      move_thread_flag_4306 = 0
      move_thread_han_4306 = run move_thread_4306()
      while (True):
        sleep(1.0E-10)
        if (move_thread_flag_4306 > 1):
          join move_thread_han_4306
          $ 4307 "Until (distance)"
          break
        end
        sync()
      end
      $ 4308 "Direction: Base Z-"
      global move_thread_flag_4308=0
      thread move_thread_4308():
        enter_critical
        move_thread_flag_4308 = 1
        local towardsPos=calculate_point_to_move_towards(p[0.0,0.0,0.0,0.0,0.0,0.0], [0.0,0.0,-1.0], 1000.0)
        movel(towardsPos, a=0.007, v=0.007)
        move_thread_flag_4308 = 2
        exit_critical
      end
      move_thread_flag_4308 = 0
      move_thread_han_4308 = run move_thread_4308()
      while (True):
        local targetTcpDirection=get_target_tcp_speed()
        local stepsToRetract=tool_contact(direction=targetTcpDirection)
        if (stepsToRetract > 0):
          kill move_thread_han_4308
          stopl(0.02)
          local backTrackMovement=get_actual_joint_positions_history(stepsToRetract)
          local contactPose=get_forward_kin(backTrackMovement)
          local posDir=[targetTcpDirection[0],targetTcpDirection[1],targetTcpDirection[2]]
          local retractTo=contactPose
          if (norm(posDir) > 1e-6):
            local normalizedPosDir=normalize(posDir)
            local additionalRetraction=p[normalizedPosDir[0] * 0.0, normalizedPosDir[1] * 0.0, normalizedPosDir[2] * 0.0, 0, 0, 0]
            retractTo = pose_sub(contactPose, additionalRetraction)
          end
          movel(retractTo, a=0.02, v=0.1)
          $ 4309 "Until (tool_contact_detection)"
          break
        end
        sync()
      end
      $ 4310 "Popup: punto contacto alanzdo"
      popup("punto contacto alanzdo", "Mensaje", False, False, blocking=True)
      $ 4311 "Direction: Base Z+"
      global move_thread_flag_4311=0
      thread move_thread_4311():
        enter_critical
        move_thread_flag_4311 = 1
        local towardsPos=calculate_point_to_move_towards(p[0.0,0.0,0.0,0.0,0.0,0.0], [0.0,0.0,1.0], 0.007)
        movel(towardsPos, a=0.015, v=0.015)
        move_thread_flag_4311 = 2
        exit_critical
      end
      move_thread_flag_4311 = 0
      move_thread_han_4311 = run move_thread_4311()
      while (True):
        sleep(1.0E-10)
        if (move_thread_flag_4311 > 1):
          join move_thread_han_4311
          $ 4312 "Until (distance)"
          break
        end
        sync()
      end
      $ 4313 "Wait: 0.3"
      sleep(0.3)
      $ 4314 "Set CO[1]=Encender"
      set_configurable_digital_out(1, True)
      $ 4315 "Wait: 0.3"
      sleep(0.3)
      $ 4316 "Loop 1 times"
      Loop_32 = 0
      while (Loop_32 < 1):
        $ 4317 "bajar≔pose_add(get_actual_tcp_pose(), bajada_broca)"
        global bajar= pose_add ( get_actual_tcp_pose (), bajada_broca)
        $ 4318 "bajar" "breakAfter"
        movel(bajar, a=0.004, v=0.004)
        $ 4319 "subir≔pose_sub(get_actual_tcp_pose(), bajada_broca)"
        global subir= pose_sub ( get_actual_tcp_pose (), bajada_broca)
        $ 4320 "Direction: Base Z+"
        global move_thread_flag_4320=0
        thread move_thread_4320():
          enter_critical
          move_thread_flag_4320 = 1
          local towardsPos=calculate_point_to_move_towards(p[0.0,0.0,0.0,0.0,0.0,0.0], [0.0,0.0,1.0], 0.002)
          movel(towardsPos, a=0.015, v=0.015)
          move_thread_flag_4320 = 2
          exit_critical
        end
        move_thread_flag_4320 = 0
        move_thread_han_4320 = run move_thread_4320()
        while (True):
          sleep(1.0E-10)
          if (move_thread_flag_4320 > 1):
            join move_thread_han_4320
            $ 4321 "Until (distance)"
            break
          end
          sync()
        end
        $ 4322 "Set CO[1]=Apagar"
        set_configurable_digital_out(1, False)
        $ 4323 "subir" "breakAfter"
        movel(subir, a=0.015, v=0.015)
        $ 4324 "bajada_broca≔pose_sub(bajada_broca, bajada)"
        global bajada_broca= pose_sub (bajada_broca, bajada)
        Loop_32 = Loop_32 + 1
      end
      $ 4325 "Direction: Base Z+"
      global move_thread_flag_4325=0
      thread move_thread_4325():
        enter_critical
        move_thread_flag_4325 = 1
        local towardsPos=calculate_point_to_move_towards(p[0.0,0.0,0.0,0.0,0.0,0.0], [0.0,0.0,1.0], 0.08)
        movel(towardsPos, a=0.15, v=0.1)
        move_thread_flag_4325 = 2
        exit_critical
      end
      move_thread_flag_4325 = 0
      move_thread_han_4325 = run move_thread_4325()
      while (True):
        sleep(1.0E-10)
        if (move_thread_flag_4325 > 1):
          join move_thread_han_4325
          $ 4326 "Until (distance)"
          break
        end
        sync()
      end
      $ 4327 "Set CO[1]=Apagar"
      set_configurable_digital_out(1, False)
      $ 4328 "barreno_actual≔barreno_actual+1"
      global barreno_actual=barreno_actual+1
    end
    $ 4331 "Popup: Linea21B con chica Terminada!"
    popup("Linea21B con chica Terminada!", "Mensaje", False, False, blocking=True)
    $ 4332 "Linea22"
    $ 4333 "Marcar_puntos"
    $ 4334 "MoveL"
    $ 4335 "Linea22_A" "breakAfter"
    movel(Linea22_A_p, a=0.5, v=0.1)
    $ 4336 "bajada_comprobacion"
    $ 4337 "Direction: Base Z-"
    global move_thread_flag_4337=0
    thread move_thread_4337():
      enter_critical
      move_thread_flag_4337 = 1
      local towardsPos=calculate_point_to_move_towards(p[0.0,0.0,0.0,0.0,0.0,0.0], [0.0,0.0,-1.0], 0.071)
      movel(towardsPos, a=0.15, v=0.1)
      move_thread_flag_4337 = 2
      exit_critical
    end
    move_thread_flag_4337 = 0
    move_thread_han_4337 = run move_thread_4337()
    while (True):
      sleep(1.0E-10)
      if (move_thread_flag_4337 > 1):
        join move_thread_han_4337
        $ 4338 "Until (distance)"
        break
      end
      sync()
    end
    $ 4339 "Direction: Base Z-"
    global move_thread_flag_4339=0
    thread move_thread_4339():
      enter_critical
      move_thread_flag_4339 = 1
      local towardsPos=calculate_point_to_move_towards(p[0.0,0.0,0.0,0.0,0.0,0.0], [0.0,0.0,-1.0], 1000.0)
      movel(towardsPos, a=0.007, v=0.007)
      move_thread_flag_4339 = 2
      exit_critical
    end
    move_thread_flag_4339 = 0
    move_thread_han_4339 = run move_thread_4339()
    while (True):
      local targetTcpDirection=get_target_tcp_speed()
      local stepsToRetract=tool_contact(direction=targetTcpDirection)
      if (stepsToRetract > 0):
        kill move_thread_han_4339
        stopl(0.02)
        local backTrackMovement=get_actual_joint_positions_history(stepsToRetract)
        local contactPose=get_forward_kin(backTrackMovement)
        local posDir=[targetTcpDirection[0],targetTcpDirection[1],targetTcpDirection[2]]
        local retractTo=contactPose
        if (norm(posDir) > 1e-6):
          local normalizedPosDir=normalize(posDir)
          local additionalRetraction=p[normalizedPosDir[0] * 0.0, normalizedPosDir[1] * 0.0, normalizedPosDir[2] * 0.0, 0, 0, 0]
          retractTo = pose_sub(contactPose, additionalRetraction)
        end
        movel(retractTo, a=0.02, v=0.1)
        $ 4340 "Until (tool_contact_detection)"
        break
      end
      sync()
    end
    $ 4341 "Direction: Base Z+"
    global move_thread_flag_4341=0
    thread move_thread_4341():
      enter_critical
      move_thread_flag_4341 = 1
      local towardsPos=calculate_point_to_move_towards(p[0.0,0.0,0.0,0.0,0.0,0.0], [0.0,0.0,1.0], 0.08)
      movel(towardsPos, a=0.15, v=0.1)
      move_thread_flag_4341 = 2
      exit_critical
    end
    move_thread_flag_4341 = 0
    move_thread_han_4341 = run move_thread_4341()
    while (True):
      sleep(1.0E-10)
      if (move_thread_flag_4341 > 1):
        join move_thread_han_4341
        $ 4342 "Until (distance)"
        break
      end
      sync()
    end
    $ 4343 "Linea22_B" "breakAfter"
    movel(Linea22_B_p, a=0.5, v=0.1)
    $ 4344 "bajada_comprobacion"
    $ 4345 "Direction: Base Z-"
    global move_thread_flag_4345=0
    thread move_thread_4345():
      enter_critical
      move_thread_flag_4345 = 1
      local towardsPos=calculate_point_to_move_towards(p[0.0,0.0,0.0,0.0,0.0,0.0], [0.0,0.0,-1.0], 0.071)
      movel(towardsPos, a=0.15, v=0.1)
      move_thread_flag_4345 = 2
      exit_critical
    end
    move_thread_flag_4345 = 0
    move_thread_han_4345 = run move_thread_4345()
    while (True):
      sleep(1.0E-10)
      if (move_thread_flag_4345 > 1):
        join move_thread_han_4345
        $ 4346 "Until (distance)"
        break
      end
      sync()
    end
    $ 4347 "Direction: Base Z-"
    global move_thread_flag_4347=0
    thread move_thread_4347():
      enter_critical
      move_thread_flag_4347 = 1
      local towardsPos=calculate_point_to_move_towards(p[0.0,0.0,0.0,0.0,0.0,0.0], [0.0,0.0,-1.0], 1000.0)
      movel(towardsPos, a=0.007, v=0.007)
      move_thread_flag_4347 = 2
      exit_critical
    end
    move_thread_flag_4347 = 0
    move_thread_han_4347 = run move_thread_4347()
    while (True):
      local targetTcpDirection=get_target_tcp_speed()
      local stepsToRetract=tool_contact(direction=targetTcpDirection)
      if (stepsToRetract > 0):
        kill move_thread_han_4347
        stopl(0.02)
        local backTrackMovement=get_actual_joint_positions_history(stepsToRetract)
        local contactPose=get_forward_kin(backTrackMovement)
        local posDir=[targetTcpDirection[0],targetTcpDirection[1],targetTcpDirection[2]]
        local retractTo=contactPose
        if (norm(posDir) > 1e-6):
          local normalizedPosDir=normalize(posDir)
          local additionalRetraction=p[normalizedPosDir[0] * 0.0, normalizedPosDir[1] * 0.0, normalizedPosDir[2] * 0.0, 0, 0, 0]
          retractTo = pose_sub(contactPose, additionalRetraction)
        end
        movel(retractTo, a=0.02, v=0.1)
        $ 4348 "Until (tool_contact_detection)"
        break
      end
      sync()
    end
    $ 4349 "Direction: Base Z+"
    global move_thread_flag_4349=0
    thread move_thread_4349():
      enter_critical
      move_thread_flag_4349 = 1
      local towardsPos=calculate_point_to_move_towards(p[0.0,0.0,0.0,0.0,0.0,0.0], [0.0,0.0,1.0], 0.08)
      movel(towardsPos, a=0.15, v=0.1)
      move_thread_flag_4349 = 2
      exit_critical
    end
    move_thread_flag_4349 = 0
    move_thread_han_4349 = run move_thread_4349()
    while (True):
      sleep(1.0E-10)
      if (move_thread_flag_4349 > 1):
        join move_thread_han_4349
        $ 4350 "Until (distance)"
        break
      end
      sync()
    end
    $ 4351 "AB"
    $ 4352 "'desbaste_inicial'"
    # 'desbaste_inicial'
    $ 4353 "bajada_broca≔p[0,0,-0.008,0,0,0]"
    global bajada_broca=p[0,0,-0.008,0,0,0]
    $ 4354 "barrenos_menos1≔1"
    global barrenos_menos1=1
    $ 4355 "barreno_actual≔0"
    global barreno_actual=0
    $ 4356 "Loop barreno_actual≤barrenos_menos1"
    while (barreno_actual <= barrenos_menos1):
      $ 4357 "Perforacion"
      $ 4358 "MoveL"
      $ 4361 "internos≔interpolate_pose(Linea22_A, Linea22_B, barreno_actual/barrenos_menos1)"
      global internos= interpolate_pose (Linea22_A_p, Linea22_B_p, barreno_actual/barrenos_menos1)
      $ 4362 "internos" "breakAfter"
      movel(internos, a=0.5, v=0.1)
      $ 4363 "'desbaste_inicial'"
      # 'desbaste_inicial'
      $ 4364 "bajada_broca≔p[0,0,-0.024,0,0,0]"
      global bajada_broca=p[0,0,-0.024,0,0,0]
      $ 4365 "bajada≔p[0,0,0.024,0,0,0]"
      global bajada=p[0,0,0.024,0,0,0]
      $ 4366 "Direction: Base Z-"
      global move_thread_flag_4366=0
      thread move_thread_4366():
        enter_critical
        move_thread_flag_4366 = 1
        local towardsPos=calculate_point_to_move_towards(p[0.0,0.0,0.0,0.0,0.0,0.0], [0.0,0.0,-1.0], 0.071)
        movel(towardsPos, a=0.15, v=0.1)
        move_thread_flag_4366 = 2
        exit_critical
      end
      move_thread_flag_4366 = 0
      move_thread_han_4366 = run move_thread_4366()
      while (True):
        sleep(1.0E-10)
        if (move_thread_flag_4366 > 1):
          join move_thread_han_4366
          $ 4367 "Until (distance)"
          break
        end
        sync()
      end
      $ 4368 "Direction: Base Z-"
      global move_thread_flag_4368=0
      thread move_thread_4368():
        enter_critical
        move_thread_flag_4368 = 1
        local towardsPos=calculate_point_to_move_towards(p[0.0,0.0,0.0,0.0,0.0,0.0], [0.0,0.0,-1.0], 1000.0)
        movel(towardsPos, a=0.007, v=0.007)
        move_thread_flag_4368 = 2
        exit_critical
      end
      move_thread_flag_4368 = 0
      move_thread_han_4368 = run move_thread_4368()
      while (True):
        local targetTcpDirection=get_target_tcp_speed()
        local stepsToRetract=tool_contact(direction=targetTcpDirection)
        if (stepsToRetract > 0):
          kill move_thread_han_4368
          stopl(0.02)
          local backTrackMovement=get_actual_joint_positions_history(stepsToRetract)
          local contactPose=get_forward_kin(backTrackMovement)
          local posDir=[targetTcpDirection[0],targetTcpDirection[1],targetTcpDirection[2]]
          local retractTo=contactPose
          if (norm(posDir) > 1e-6):
            local normalizedPosDir=normalize(posDir)
            local additionalRetraction=p[normalizedPosDir[0] * 0.0, normalizedPosDir[1] * 0.0, normalizedPosDir[2] * 0.0, 0, 0, 0]
            retractTo = pose_sub(contactPose, additionalRetraction)
          end
          movel(retractTo, a=0.02, v=0.1)
          $ 4369 "Until (tool_contact_detection)"
          break
        end
        sync()
      end
      $ 4370 "Popup: punto contacto alanzdo"
      popup("punto contacto alanzdo", "Mensaje", False, False, blocking=True)
      $ 4371 "Direction: Base Z+"
      global move_thread_flag_4371=0
      thread move_thread_4371():
        enter_critical
        move_thread_flag_4371 = 1
        local towardsPos=calculate_point_to_move_towards(p[0.0,0.0,0.0,0.0,0.0,0.0], [0.0,0.0,1.0], 0.007)
        movel(towardsPos, a=0.015, v=0.015)
        move_thread_flag_4371 = 2
        exit_critical
      end
      move_thread_flag_4371 = 0
      move_thread_han_4371 = run move_thread_4371()
      while (True):
        sleep(1.0E-10)
        if (move_thread_flag_4371 > 1):
          join move_thread_han_4371
          $ 4372 "Until (distance)"
          break
        end
        sync()
      end
      $ 4373 "Wait: 0.3"
      sleep(0.3)
      $ 4374 "Set CO[1]=Encender"
      set_configurable_digital_out(1, True)
      $ 4375 "Wait: 0.3"
      sleep(0.3)
      $ 4376 "Loop 1 times"
      Loop_84 = 0
      while (Loop_84 < 1):
        $ 4377 "bajar≔pose_add(get_actual_tcp_pose(), bajada_broca)"
        global bajar= pose_add ( get_actual_tcp_pose (), bajada_broca)
        $ 4378 "bajar" "breakAfter"
        movel(bajar, a=0.004, v=0.004)
        $ 4379 "subir≔pose_sub(get_actual_tcp_pose(), bajada_broca)"
        global subir= pose_sub ( get_actual_tcp_pose (), bajada_broca)
        $ 4380 "Direction: Base Z+"
        global move_thread_flag_4380=0
        thread move_thread_4380():
          enter_critical
          move_thread_flag_4380 = 1
          local towardsPos=calculate_point_to_move_towards(p[0.0,0.0,0.0,0.0,0.0,0.0], [0.0,0.0,1.0], 0.002)
          movel(towardsPos, a=0.015, v=0.015)
          move_thread_flag_4380 = 2
          exit_critical
        end
        move_thread_flag_4380 = 0
        move_thread_han_4380 = run move_thread_4380()
        while (True):
          sleep(1.0E-10)
          if (move_thread_flag_4380 > 1):
            join move_thread_han_4380
            $ 4381 "Until (distance)"
            break
          end
          sync()
        end
        $ 4382 "Set CO[1]=Apagar"
        set_configurable_digital_out(1, False)
        $ 4383 "subir" "breakAfter"
        movel(subir, a=0.01, v=0.005)
        $ 4384 "bajada_broca≔pose_sub(bajada_broca, bajada)"
        global bajada_broca= pose_sub (bajada_broca, bajada)
        Loop_84 = Loop_84 + 1
      end
      $ 4385 "Direction: Base Z+"
      global move_thread_flag_4385=0
      thread move_thread_4385():
        enter_critical
        move_thread_flag_4385 = 1
        local towardsPos=calculate_point_to_move_towards(p[0.0,0.0,0.0,0.0,0.0,0.0], [0.0,0.0,1.0], 0.08)
        movel(towardsPos, a=0.15, v=0.1)
        move_thread_flag_4385 = 2
        exit_critical
      end
      move_thread_flag_4385 = 0
      move_thread_han_4385 = run move_thread_4385()
      while (True):
        sleep(1.0E-10)
        if (move_thread_flag_4385 > 1):
          join move_thread_han_4385
          $ 4386 "Until (distance)"
          break
        end
        sync()
      end
      $ 4387 "Set CO[1]=Apagar"
      set_configurable_digital_out(1, False)
      $ 4388 "barreno_actual≔barreno_actual+1"
      global barreno_actual=barreno_actual+1
    end
    $ 4391 "Popup: Linea22 con chica Terminada!"
    popup("Linea22 con chica Terminada!", "Mensaje", False, False, blocking=True)
    $ 4392 "Linea23"
    $ 4393 "Marcar_puntos"
    $ 4394 "MoveL"
    $ 4395 "Linea23_A" "breakAfter"
    movel(Linea23_A_p, a=0.5, v=0.1)
    $ 4396 "bajada_comprobacion"
    $ 4397 "Direction: Base Z-"
    global move_thread_flag_4397=0
    thread move_thread_4397():
      enter_critical
      move_thread_flag_4397 = 1
      local towardsPos=calculate_point_to_move_towards(p[0.0,0.0,0.0,0.0,0.0,0.0], [0.0,0.0,-1.0], 0.071)
      movel(towardsPos, a=0.15, v=0.1)
      move_thread_flag_4397 = 2
      exit_critical
    end
    move_thread_flag_4397 = 0
    move_thread_han_4397 = run move_thread_4397()
    while (True):
      sleep(1.0E-10)
      if (move_thread_flag_4397 > 1):
        join move_thread_han_4397
        $ 4398 "Until (distance)"
        break
      end
      sync()
    end
    $ 4399 "Direction: Base Z-"
    global move_thread_flag_4399=0
    thread move_thread_4399():
      enter_critical
      move_thread_flag_4399 = 1
      local towardsPos=calculate_point_to_move_towards(p[0.0,0.0,0.0,0.0,0.0,0.0], [0.0,0.0,-1.0], 1000.0)
      movel(towardsPos, a=0.007, v=0.007)
      move_thread_flag_4399 = 2
      exit_critical
    end
    move_thread_flag_4399 = 0
    move_thread_han_4399 = run move_thread_4399()
    while (True):
      local targetTcpDirection=get_target_tcp_speed()
      local stepsToRetract=tool_contact(direction=targetTcpDirection)
      if (stepsToRetract > 0):
        kill move_thread_han_4399
        stopl(0.02)
        local backTrackMovement=get_actual_joint_positions_history(stepsToRetract)
        local contactPose=get_forward_kin(backTrackMovement)
        local posDir=[targetTcpDirection[0],targetTcpDirection[1],targetTcpDirection[2]]
        local retractTo=contactPose
        if (norm(posDir) > 1e-6):
          local normalizedPosDir=normalize(posDir)
          local additionalRetraction=p[normalizedPosDir[0] * 0.0, normalizedPosDir[1] * 0.0, normalizedPosDir[2] * 0.0, 0, 0, 0]
          retractTo = pose_sub(contactPose, additionalRetraction)
        end
        movel(retractTo, a=0.02, v=0.1)
        $ 4400 "Until (tool_contact_detection)"
        break
      end
      sync()
    end
    $ 4401 "Direction: Base Z+"
    global move_thread_flag_4401=0
    thread move_thread_4401():
      enter_critical
      move_thread_flag_4401 = 1
      local towardsPos=calculate_point_to_move_towards(p[0.0,0.0,0.0,0.0,0.0,0.0], [0.0,0.0,1.0], 0.08)
      movel(towardsPos, a=0.15, v=0.1)
      move_thread_flag_4401 = 2
      exit_critical
    end
    move_thread_flag_4401 = 0
    move_thread_han_4401 = run move_thread_4401()
    while (True):
      sleep(1.0E-10)
      if (move_thread_flag_4401 > 1):
        join move_thread_han_4401
        $ 4402 "Until (distance)"
        break
      end
      sync()
    end
    $ 4403 "Linea23_B" "breakAfter"
    movel(Linea23_B_p, a=0.5, v=0.1)
    $ 4404 "bajada_comprobacion"
    $ 4405 "Direction: Base Z-"
    global move_thread_flag_4405=0
    thread move_thread_4405():
      enter_critical
      move_thread_flag_4405 = 1
      local towardsPos=calculate_point_to_move_towards(p[0.0,0.0,0.0,0.0,0.0,0.0], [0.0,0.0,-1.0], 0.071)
      movel(towardsPos, a=0.15, v=0.1)
      move_thread_flag_4405 = 2
      exit_critical
    end
    move_thread_flag_4405 = 0
    move_thread_han_4405 = run move_thread_4405()
    while (True):
      sleep(1.0E-10)
      if (move_thread_flag_4405 > 1):
        join move_thread_han_4405
        $ 4406 "Until (distance)"
        break
      end
      sync()
    end
    $ 4407 "Direction: Base Z-"
    global move_thread_flag_4407=0
    thread move_thread_4407():
      enter_critical
      move_thread_flag_4407 = 1
      local towardsPos=calculate_point_to_move_towards(p[0.0,0.0,0.0,0.0,0.0,0.0], [0.0,0.0,-1.0], 1000.0)
      movel(towardsPos, a=0.007, v=0.007)
      move_thread_flag_4407 = 2
      exit_critical
    end
    move_thread_flag_4407 = 0
    move_thread_han_4407 = run move_thread_4407()
    while (True):
      local targetTcpDirection=get_target_tcp_speed()
      local stepsToRetract=tool_contact(direction=targetTcpDirection)
      if (stepsToRetract > 0):
        kill move_thread_han_4407
        stopl(0.02)
        local backTrackMovement=get_actual_joint_positions_history(stepsToRetract)
        local contactPose=get_forward_kin(backTrackMovement)
        local posDir=[targetTcpDirection[0],targetTcpDirection[1],targetTcpDirection[2]]
        local retractTo=contactPose
        if (norm(posDir) > 1e-6):
          local normalizedPosDir=normalize(posDir)
          local additionalRetraction=p[normalizedPosDir[0] * 0.0, normalizedPosDir[1] * 0.0, normalizedPosDir[2] * 0.0, 0, 0, 0]
          retractTo = pose_sub(contactPose, additionalRetraction)
        end
        movel(retractTo, a=0.02, v=0.1)
        $ 4408 "Until (tool_contact_detection)"
        break
      end
      sync()
    end
    $ 4409 "Direction: Base Z+"
    global move_thread_flag_4409=0
    thread move_thread_4409():
      enter_critical
      move_thread_flag_4409 = 1
      local towardsPos=calculate_point_to_move_towards(p[0.0,0.0,0.0,0.0,0.0,0.0], [0.0,0.0,1.0], 0.08)
      movel(towardsPos, a=0.15, v=0.1)
      move_thread_flag_4409 = 2
      exit_critical
    end
    move_thread_flag_4409 = 0
    move_thread_han_4409 = run move_thread_4409()
    while (True):
      sleep(1.0E-10)
      if (move_thread_flag_4409 > 1):
        join move_thread_han_4409
        $ 4410 "Until (distance)"
        break
      end
      sync()
    end
    $ 4411 "AB"
    $ 4412 "'desbaste_inicial'"
    # 'desbaste_inicial'
    $ 4413 "bajada_broca≔p[0,0,-0.008,0,0,0]"
    global bajada_broca=p[0,0,-0.008,0,0,0]
    $ 4414 "barrenos_menos1≔2"
    global barrenos_menos1=2
    $ 4415 "barreno_actual≔0"
    global barreno_actual=0
    $ 4416 "Loop barreno_actual≤barrenos_menos1"
    while (barreno_actual <= barrenos_menos1):
      $ 4417 "Perforacion"
      $ 4418 "MoveL"
      $ 4421 "internos≔interpolate_pose(Linea23_A, Linea23_B, barreno_actual/barrenos_menos1)"
      global internos= interpolate_pose (Linea23_A_p, Linea23_B_p, barreno_actual/barrenos_menos1)
      $ 4422 "internos" "breakAfter"
      movel(internos, a=0.5, v=0.1)
      $ 4423 "'desbaste_inicial'"
      # 'desbaste_inicial'
      $ 4424 "bajada_broca≔p[0,0,-0.024,0,0,0]"
      global bajada_broca=p[0,0,-0.024,0,0,0]
      $ 4425 "bajada≔p[0,0,0.024,0,0,0]"
      global bajada=p[0,0,0.024,0,0,0]
      $ 4426 "Direction: Base Z-"
      global move_thread_flag_4426=0
      thread move_thread_4426():
        enter_critical
        move_thread_flag_4426 = 1
        local towardsPos=calculate_point_to_move_towards(p[0.0,0.0,0.0,0.0,0.0,0.0], [0.0,0.0,-1.0], 0.071)
        movel(towardsPos, a=0.15, v=0.1)
        move_thread_flag_4426 = 2
        exit_critical
      end
      move_thread_flag_4426 = 0
      move_thread_han_4426 = run move_thread_4426()
      while (True):
        sleep(1.0E-10)
        if (move_thread_flag_4426 > 1):
          join move_thread_han_4426
          $ 4427 "Until (distance)"
          break
        end
        sync()
      end
      $ 4428 "Direction: Base Z-"
      global move_thread_flag_4428=0
      thread move_thread_4428():
        enter_critical
        move_thread_flag_4428 = 1
        local towardsPos=calculate_point_to_move_towards(p[0.0,0.0,0.0,0.0,0.0,0.0], [0.0,0.0,-1.0], 1000.0)
        movel(towardsPos, a=0.007, v=0.007)
        move_thread_flag_4428 = 2
        exit_critical
      end
      move_thread_flag_4428 = 0
      move_thread_han_4428 = run move_thread_4428()
      while (True):
        local targetTcpDirection=get_target_tcp_speed()
        local stepsToRetract=tool_contact(direction=targetTcpDirection)
        if (stepsToRetract > 0):
          kill move_thread_han_4428
          stopl(0.02)
          local backTrackMovement=get_actual_joint_positions_history(stepsToRetract)
          local contactPose=get_forward_kin(backTrackMovement)
          local posDir=[targetTcpDirection[0],targetTcpDirection[1],targetTcpDirection[2]]
          local retractTo=contactPose
          if (norm(posDir) > 1e-6):
            local normalizedPosDir=normalize(posDir)
            local additionalRetraction=p[normalizedPosDir[0] * 0.0, normalizedPosDir[1] * 0.0, normalizedPosDir[2] * 0.0, 0, 0, 0]
            retractTo = pose_sub(contactPose, additionalRetraction)
          end
          movel(retractTo, a=0.02, v=0.1)
          $ 4429 "Until (tool_contact_detection)"
          break
        end
        sync()
      end
      $ 4430 "Popup: punto contacto alanzdo"
      popup("punto contacto alanzdo", "Mensaje", False, False, blocking=True)
      $ 4431 "Direction: Base Z+"
      global move_thread_flag_4431=0
      thread move_thread_4431():
        enter_critical
        move_thread_flag_4431 = 1
        local towardsPos=calculate_point_to_move_towards(p[0.0,0.0,0.0,0.0,0.0,0.0], [0.0,0.0,1.0], 0.007)
        movel(towardsPos, a=0.015, v=0.015)
        move_thread_flag_4431 = 2
        exit_critical
      end
      move_thread_flag_4431 = 0
      move_thread_han_4431 = run move_thread_4431()
      while (True):
        sleep(1.0E-10)
        if (move_thread_flag_4431 > 1):
          join move_thread_han_4431
          $ 4432 "Until (distance)"
          break
        end
        sync()
      end
      $ 4433 "Wait: 0.3"
      sleep(0.3)
      $ 4434 "Set CO[1]=Encender"
      set_configurable_digital_out(1, True)
      $ 4435 "Wait: 0.3"
      sleep(0.3)
      $ 4436 "Loop 1 times"
      Loop_88 = 0
      while (Loop_88 < 1):
        $ 4437 "bajar≔pose_add(get_actual_tcp_pose(), bajada_broca)"
        global bajar= pose_add ( get_actual_tcp_pose (), bajada_broca)
        $ 4438 "bajar" "breakAfter"
        movel(bajar, a=0.004, v=0.004)
        $ 4439 "subir≔pose_sub(get_actual_tcp_pose(), bajada_broca)"
        global subir= pose_sub ( get_actual_tcp_pose (), bajada_broca)
        $ 4440 "Direction: Base Z+"
        global move_thread_flag_4440=0
        thread move_thread_4440():
          enter_critical
          move_thread_flag_4440 = 1
          local towardsPos=calculate_point_to_move_towards(p[0.0,0.0,0.0,0.0,0.0,0.0], [0.0,0.0,1.0], 0.002)
          movel(towardsPos, a=0.015, v=0.015)
          move_thread_flag_4440 = 2
          exit_critical
        end
        move_thread_flag_4440 = 0
        move_thread_han_4440 = run move_thread_4440()
        while (True):
          sleep(1.0E-10)
          if (move_thread_flag_4440 > 1):
            join move_thread_han_4440
            $ 4441 "Until (distance)"
            break
          end
          sync()
        end
        $ 4442 "Set CO[1]=Apagar"
        set_configurable_digital_out(1, False)
        $ 4443 "subir" "breakAfter"
        movel(subir, a=0.015, v=0.015)
        $ 4444 "bajada_broca≔pose_sub(bajada_broca, bajada)"
        global bajada_broca= pose_sub (bajada_broca, bajada)
        Loop_88 = Loop_88 + 1
      end
      $ 4445 "Direction: Base Z+"
      global move_thread_flag_4445=0
      thread move_thread_4445():
        enter_critical
        move_thread_flag_4445 = 1
        local towardsPos=calculate_point_to_move_towards(p[0.0,0.0,0.0,0.0,0.0,0.0], [0.0,0.0,1.0], 0.08)
        movel(towardsPos, a=0.15, v=0.1)
        move_thread_flag_4445 = 2
        exit_critical
      end
      move_thread_flag_4445 = 0
      move_thread_han_4445 = run move_thread_4445()
      while (True):
        sleep(1.0E-10)
        if (move_thread_flag_4445 > 1):
          join move_thread_han_4445
          $ 4446 "Until (distance)"
          break
        end
        sync()
      end
      $ 4447 "Set CO[1]=Apagar"
      set_configurable_digital_out(1, False)
      $ 4448 "barreno_actual≔barreno_actual+1"
      global barreno_actual=barreno_actual+1
    end
    $ 4451 "Popup: Linea23 con chica Terminada!"
    popup("Linea23 con chica Terminada!", "Mensaje", False, False, blocking=True)
    $ 4452 "Linea24"
    $ 4453 "Marcar_puntos"
    $ 4454 "MoveL"
    $ 4455 "Linea24_A" "breakAfter"
    movel(Linea24_A_p, a=0.5, v=0.1)
    $ 4456 "bajada_comprobacion"
    $ 4457 "Direction: Base Z-"
    global move_thread_flag_4457=0
    thread move_thread_4457():
      enter_critical
      move_thread_flag_4457 = 1
      local towardsPos=calculate_point_to_move_towards(p[0.0,0.0,0.0,0.0,0.0,0.0], [0.0,0.0,-1.0], 0.071)
      movel(towardsPos, a=0.15, v=0.1)
      move_thread_flag_4457 = 2
      exit_critical
    end
    move_thread_flag_4457 = 0
    move_thread_han_4457 = run move_thread_4457()
    while (True):
      sleep(1.0E-10)
      if (move_thread_flag_4457 > 1):
        join move_thread_han_4457
        $ 4458 "Until (distance)"
        break
      end
      sync()
    end
    $ 4459 "Direction: Base Z-"
    global move_thread_flag_4459=0
    thread move_thread_4459():
      enter_critical
      move_thread_flag_4459 = 1
      local towardsPos=calculate_point_to_move_towards(p[0.0,0.0,0.0,0.0,0.0,0.0], [0.0,0.0,-1.0], 1000.0)
      movel(towardsPos, a=0.007, v=0.007)
      move_thread_flag_4459 = 2
      exit_critical
    end
    move_thread_flag_4459 = 0
    move_thread_han_4459 = run move_thread_4459()
    while (True):
      local targetTcpDirection=get_target_tcp_speed()
      local stepsToRetract=tool_contact(direction=targetTcpDirection)
      if (stepsToRetract > 0):
        kill move_thread_han_4459
        stopl(0.02)
        local backTrackMovement=get_actual_joint_positions_history(stepsToRetract)
        local contactPose=get_forward_kin(backTrackMovement)
        local posDir=[targetTcpDirection[0],targetTcpDirection[1],targetTcpDirection[2]]
        local retractTo=contactPose
        if (norm(posDir) > 1e-6):
          local normalizedPosDir=normalize(posDir)
          local additionalRetraction=p[normalizedPosDir[0] * 0.0, normalizedPosDir[1] * 0.0, normalizedPosDir[2] * 0.0, 0, 0, 0]
          retractTo = pose_sub(contactPose, additionalRetraction)
        end
        movel(retractTo, a=0.02, v=0.1)
        $ 4460 "Until (tool_contact_detection)"
        break
      end
      sync()
    end
    $ 4461 "Direction: Base Z+"
    global move_thread_flag_4461=0
    thread move_thread_4461():
      enter_critical
      move_thread_flag_4461 = 1
      local towardsPos=calculate_point_to_move_towards(p[0.0,0.0,0.0,0.0,0.0,0.0], [0.0,0.0,1.0], 0.08)
      movel(towardsPos, a=0.15, v=0.1)
      move_thread_flag_4461 = 2
      exit_critical
    end
    move_thread_flag_4461 = 0
    move_thread_han_4461 = run move_thread_4461()
    while (True):
      sleep(1.0E-10)
      if (move_thread_flag_4461 > 1):
        join move_thread_han_4461
        $ 4462 "Until (distance)"
        break
      end
      sync()
    end
    $ 4463 "Linea24_B" "breakAfter"
    movel(Linea24_B_p, a=0.5, v=0.1)
    $ 4464 "bajada_comprobacion"
    $ 4465 "Direction: Base Z-"
    global move_thread_flag_4465=0
    thread move_thread_4465():
      enter_critical
      move_thread_flag_4465 = 1
      local towardsPos=calculate_point_to_move_towards(p[0.0,0.0,0.0,0.0,0.0,0.0], [0.0,0.0,-1.0], 0.071)
      movel(towardsPos, a=0.15, v=0.1)
      move_thread_flag_4465 = 2
      exit_critical
    end
    move_thread_flag_4465 = 0
    move_thread_han_4465 = run move_thread_4465()
    while (True):
      sleep(1.0E-10)
      if (move_thread_flag_4465 > 1):
        join move_thread_han_4465
        $ 4466 "Until (distance)"
        break
      end
      sync()
    end
    $ 4467 "Direction: Base Z-"
    global move_thread_flag_4467=0
    thread move_thread_4467():
      enter_critical
      move_thread_flag_4467 = 1
      local towardsPos=calculate_point_to_move_towards(p[0.0,0.0,0.0,0.0,0.0,0.0], [0.0,0.0,-1.0], 1000.0)
      movel(towardsPos, a=0.007, v=0.007)
      move_thread_flag_4467 = 2
      exit_critical
    end
    move_thread_flag_4467 = 0
    move_thread_han_4467 = run move_thread_4467()
    while (True):
      local targetTcpDirection=get_target_tcp_speed()
      local stepsToRetract=tool_contact(direction=targetTcpDirection)
      if (stepsToRetract > 0):
        kill move_thread_han_4467
        stopl(0.02)
        local backTrackMovement=get_actual_joint_positions_history(stepsToRetract)
        local contactPose=get_forward_kin(backTrackMovement)
        local posDir=[targetTcpDirection[0],targetTcpDirection[1],targetTcpDirection[2]]
        local retractTo=contactPose
        if (norm(posDir) > 1e-6):
          local normalizedPosDir=normalize(posDir)
          local additionalRetraction=p[normalizedPosDir[0] * 0.0, normalizedPosDir[1] * 0.0, normalizedPosDir[2] * 0.0, 0, 0, 0]
          retractTo = pose_sub(contactPose, additionalRetraction)
        end
        movel(retractTo, a=0.02, v=0.1)
        $ 4468 "Until (tool_contact_detection)"
        break
      end
      sync()
    end
    $ 4469 "Direction: Base Z+"
    global move_thread_flag_4469=0
    thread move_thread_4469():
      enter_critical
      move_thread_flag_4469 = 1
      local towardsPos=calculate_point_to_move_towards(p[0.0,0.0,0.0,0.0,0.0,0.0], [0.0,0.0,1.0], 0.08)
      movel(towardsPos, a=0.15, v=0.1)
      move_thread_flag_4469 = 2
      exit_critical
    end
    move_thread_flag_4469 = 0
    move_thread_han_4469 = run move_thread_4469()
    while (True):
      sleep(1.0E-10)
      if (move_thread_flag_4469 > 1):
        join move_thread_han_4469
        $ 4470 "Until (distance)"
        break
      end
      sync()
    end
    $ 4471 "AB"
    $ 4472 "'desbaste_inicial'"
    # 'desbaste_inicial'
    $ 4473 "bajada_broca≔p[0,0,-0.008,0,0,0]"
    global bajada_broca=p[0,0,-0.008,0,0,0]
    $ 4474 "barrenos_menos1≔4"
    global barrenos_menos1=4
    $ 4475 "barreno_actual≔0"
    global barreno_actual=0
    $ 4476 "Loop barreno_actual≤barrenos_menos1"
    while (barreno_actual <= barrenos_menos1):
      $ 4477 "Perforacion"
      $ 4478 "MoveL"
      $ 4479 "If barreno_actual≟2"
      if (barreno_actual == 2):
        $ 4480 "barreno_actual≔barreno_actual+1"
        global barreno_actual=barreno_actual+1
      end
      $ 4481 "internos≔interpolate_pose(Linea24_A, Linea24_B, barreno_actual/barrenos_menos1)"
      global internos= interpolate_pose (Linea24_A_p, Linea24_B_p, barreno_actual/barrenos_menos1)
      $ 4482 "internos" "breakAfter"
      movel(internos, a=0.5, v=0.1)
      $ 4483 "'desbaste_inicial'"
      # 'desbaste_inicial'
      $ 4484 "bajada_broca≔p[0,0,-0.024,0,0,0]"
      global bajada_broca=p[0,0,-0.024,0,0,0]
      $ 4485 "bajada≔p[0,0,0.024,0,0,0]"
      global bajada=p[0,0,0.024,0,0,0]
      $ 4486 "Direction: Base Z-"
      global move_thread_flag_4486=0
      thread move_thread_4486():
        enter_critical
        move_thread_flag_4486 = 1
        local towardsPos=calculate_point_to_move_towards(p[0.0,0.0,0.0,0.0,0.0,0.0], [0.0,0.0,-1.0], 0.071)
        movel(towardsPos, a=0.15, v=0.1)
        move_thread_flag_4486 = 2
        exit_critical
      end
      move_thread_flag_4486 = 0
      move_thread_han_4486 = run move_thread_4486()
      while (True):
        sleep(1.0E-10)
        if (move_thread_flag_4486 > 1):
          join move_thread_han_4486
          $ 4487 "Until (distance)"
          break
        end
        sync()
      end
      $ 4488 "Direction: Base Z-"
      global move_thread_flag_4488=0
      thread move_thread_4488():
        enter_critical
        move_thread_flag_4488 = 1
        local towardsPos=calculate_point_to_move_towards(p[0.0,0.0,0.0,0.0,0.0,0.0], [0.0,0.0,-1.0], 1000.0)
        movel(towardsPos, a=0.007, v=0.007)
        move_thread_flag_4488 = 2
        exit_critical
      end
      move_thread_flag_4488 = 0
      move_thread_han_4488 = run move_thread_4488()
      while (True):
        local targetTcpDirection=get_target_tcp_speed()
        local stepsToRetract=tool_contact(direction=targetTcpDirection)
        if (stepsToRetract > 0):
          kill move_thread_han_4488
          stopl(0.02)
          local backTrackMovement=get_actual_joint_positions_history(stepsToRetract)
          local contactPose=get_forward_kin(backTrackMovement)
          local posDir=[targetTcpDirection[0],targetTcpDirection[1],targetTcpDirection[2]]
          local retractTo=contactPose
          if (norm(posDir) > 1e-6):
            local normalizedPosDir=normalize(posDir)
            local additionalRetraction=p[normalizedPosDir[0] * 0.0, normalizedPosDir[1] * 0.0, normalizedPosDir[2] * 0.0, 0, 0, 0]
            retractTo = pose_sub(contactPose, additionalRetraction)
          end
          movel(retractTo, a=0.02, v=0.1)
          $ 4489 "Until (tool_contact_detection)"
          break
        end
        sync()
      end
      $ 4490 "Popup: punto contacto alanzdo"
      popup("punto contacto alanzdo", "Mensaje", False, False, blocking=True)
      $ 4491 "Direction: Base Z+"
      global move_thread_flag_4491=0
      thread move_thread_4491():
        enter_critical
        move_thread_flag_4491 = 1
        local towardsPos=calculate_point_to_move_towards(p[0.0,0.0,0.0,0.0,0.0,0.0], [0.0,0.0,1.0], 0.007)
        movel(towardsPos, a=0.015, v=0.015)
        move_thread_flag_4491 = 2
        exit_critical
      end
      move_thread_flag_4491 = 0
      move_thread_han_4491 = run move_thread_4491()
      while (True):
        sleep(1.0E-10)
        if (move_thread_flag_4491 > 1):
          join move_thread_han_4491
          $ 4492 "Until (distance)"
          break
        end
        sync()
      end
      $ 4493 "Wait: 0.3"
      sleep(0.3)
      $ 4494 "Set CO[1]=Encender"
      set_configurable_digital_out(1, True)
      $ 4495 "Wait: 0.3"
      sleep(0.3)
      $ 4496 "Loop 1 times"
      Loop_102 = 0
      while (Loop_102 < 1):
        $ 4497 "bajar≔pose_add(get_actual_tcp_pose(), bajada_broca)"
        global bajar= pose_add ( get_actual_tcp_pose (), bajada_broca)
        $ 4498 "bajar" "breakAfter"
        movel(bajar, a=0.004, v=0.004)
        $ 4499 "subir≔pose_sub(get_actual_tcp_pose(), bajada_broca)"
        global subir= pose_sub ( get_actual_tcp_pose (), bajada_broca)
        $ 4500 "Direction: Base Z+"
        global move_thread_flag_4500=0
        thread move_thread_4500():
          enter_critical
          move_thread_flag_4500 = 1
          local towardsPos=calculate_point_to_move_towards(p[0.0,0.0,0.0,0.0,0.0,0.0], [0.0,0.0,1.0], 0.002)
          movel(towardsPos, a=0.015, v=0.015)
          move_thread_flag_4500 = 2
          exit_critical
        end
        move_thread_flag_4500 = 0
        move_thread_han_4500 = run move_thread_4500()
        while (True):
          sleep(1.0E-10)
          if (move_thread_flag_4500 > 1):
            join move_thread_han_4500
            $ 4501 "Until (distance)"
            break
          end
          sync()
        end
        $ 4502 "Set CO[1]=Apagar"
        set_configurable_digital_out(1, False)
        $ 4503 "subir" "breakAfter"
        movel(subir, a=0.015, v=0.015)
        $ 4504 "bajada_broca≔pose_sub(bajada_broca, bajada)"
        global bajada_broca= pose_sub (bajada_broca, bajada)
        Loop_102 = Loop_102 + 1
      end
      $ 4505 "Direction: Base Z+"
      global move_thread_flag_4505=0
      thread move_thread_4505():
        enter_critical
        move_thread_flag_4505 = 1
        local towardsPos=calculate_point_to_move_towards(p[0.0,0.0,0.0,0.0,0.0,0.0], [0.0,0.0,1.0], 0.08)
        movel(towardsPos, a=0.15, v=0.1)
        move_thread_flag_4505 = 2
        exit_critical
      end
      move_thread_flag_4505 = 0
      move_thread_han_4505 = run move_thread_4505()
      while (True):
        sleep(1.0E-10)
        if (move_thread_flag_4505 > 1):
          join move_thread_han_4505
          $ 4506 "Until (distance)"
          break
        end
        sync()
      end
      $ 4507 "Set CO[1]=Apagar"
      set_configurable_digital_out(1, False)
      $ 4508 "barreno_actual≔barreno_actual+1"
      global barreno_actual=barreno_actual+1
    end
    $ 4511 "Popup: Linea24 con chica Terminada!"
    popup("Linea24 con chica Terminada!", "Mensaje", False, False, blocking=True)
    $ 4512 "Linea25"
    $ 4513 "Marcar_puntos"
    $ 4514 "MoveL"
    $ 4515 "Linea25_A" "breakAfter"
    movel(Linea25_A_p, a=0.5, v=0.1)
    $ 4516 "bajada_comprobacion"
    $ 4517 "Direction: Base Z-"
    global move_thread_flag_4517=0
    thread move_thread_4517():
      enter_critical
      move_thread_flag_4517 = 1
      local towardsPos=calculate_point_to_move_towards(p[0.0,0.0,0.0,0.0,0.0,0.0], [0.0,0.0,-1.0], 0.071)
      movel(towardsPos, a=0.15, v=0.1)
      move_thread_flag_4517 = 2
      exit_critical
    end
    move_thread_flag_4517 = 0
    move_thread_han_4517 = run move_thread_4517()
    while (True):
      sleep(1.0E-10)
      if (move_thread_flag_4517 > 1):
        join move_thread_han_4517
        $ 4518 "Until (distance)"
        break
      end
      sync()
    end
    $ 4519 "Direction: Base Z-"
    global move_thread_flag_4519=0
    thread move_thread_4519():
      enter_critical
      move_thread_flag_4519 = 1
      local towardsPos=calculate_point_to_move_towards(p[0.0,0.0,0.0,0.0,0.0,0.0], [0.0,0.0,-1.0], 1000.0)
      movel(towardsPos, a=0.007, v=0.007)
      move_thread_flag_4519 = 2
      exit_critical
    end
    move_thread_flag_4519 = 0
    move_thread_han_4519 = run move_thread_4519()
    while (True):
      local targetTcpDirection=get_target_tcp_speed()
      local stepsToRetract=tool_contact(direction=targetTcpDirection)
      if (stepsToRetract > 0):
        kill move_thread_han_4519
        stopl(0.02)
        local backTrackMovement=get_actual_joint_positions_history(stepsToRetract)
        local contactPose=get_forward_kin(backTrackMovement)
        local posDir=[targetTcpDirection[0],targetTcpDirection[1],targetTcpDirection[2]]
        local retractTo=contactPose
        if (norm(posDir) > 1e-6):
          local normalizedPosDir=normalize(posDir)
          local additionalRetraction=p[normalizedPosDir[0] * 0.0, normalizedPosDir[1] * 0.0, normalizedPosDir[2] * 0.0, 0, 0, 0]
          retractTo = pose_sub(contactPose, additionalRetraction)
        end
        movel(retractTo, a=0.02, v=0.1)
        $ 4520 "Until (tool_contact_detection)"
        break
      end
      sync()
    end
    $ 4521 "Direction: Base Z+"
    global move_thread_flag_4521=0
    thread move_thread_4521():
      enter_critical
      move_thread_flag_4521 = 1
      local towardsPos=calculate_point_to_move_towards(p[0.0,0.0,0.0,0.0,0.0,0.0], [0.0,0.0,1.0], 0.08)
      movel(towardsPos, a=0.15, v=0.1)
      move_thread_flag_4521 = 2
      exit_critical
    end
    move_thread_flag_4521 = 0
    move_thread_han_4521 = run move_thread_4521()
    while (True):
      sleep(1.0E-10)
      if (move_thread_flag_4521 > 1):
        join move_thread_han_4521
        $ 4522 "Until (distance)"
        break
      end
      sync()
    end
    $ 4523 "Linea25_B" "breakAfter"
    movel(Linea25_B_p, a=0.5, v=0.1)
    $ 4524 "bajada_comprobacion"
    $ 4525 "Direction: Base Z-"
    global move_thread_flag_4525=0
    thread move_thread_4525():
      enter_critical
      move_thread_flag_4525 = 1
      local towardsPos=calculate_point_to_move_towards(p[0.0,0.0,0.0,0.0,0.0,0.0], [0.0,0.0,-1.0], 0.071)
      movel(towardsPos, a=0.15, v=0.1)
      move_thread_flag_4525 = 2
      exit_critical
    end
    move_thread_flag_4525 = 0
    move_thread_han_4525 = run move_thread_4525()
    while (True):
      sleep(1.0E-10)
      if (move_thread_flag_4525 > 1):
        join move_thread_han_4525
        $ 4526 "Until (distance)"
        break
      end
      sync()
    end
    $ 4527 "Direction: Base Z-"
    global move_thread_flag_4527=0
    thread move_thread_4527():
      enter_critical
      move_thread_flag_4527 = 1
      local towardsPos=calculate_point_to_move_towards(p[0.0,0.0,0.0,0.0,0.0,0.0], [0.0,0.0,-1.0], 1000.0)
      movel(towardsPos, a=0.007, v=0.007)
      move_thread_flag_4527 = 2
      exit_critical
    end
    move_thread_flag_4527 = 0
    move_thread_han_4527 = run move_thread_4527()
    while (True):
      local targetTcpDirection=get_target_tcp_speed()
      local stepsToRetract=tool_contact(direction=targetTcpDirection)
      if (stepsToRetract > 0):
        kill move_thread_han_4527
        stopl(0.02)
        local backTrackMovement=get_actual_joint_positions_history(stepsToRetract)
        local contactPose=get_forward_kin(backTrackMovement)
        local posDir=[targetTcpDirection[0],targetTcpDirection[1],targetTcpDirection[2]]
        local retractTo=contactPose
        if (norm(posDir) > 1e-6):
          local normalizedPosDir=normalize(posDir)
          local additionalRetraction=p[normalizedPosDir[0] * 0.0, normalizedPosDir[1] * 0.0, normalizedPosDir[2] * 0.0, 0, 0, 0]
          retractTo = pose_sub(contactPose, additionalRetraction)
        end
        movel(retractTo, a=0.02, v=0.1)
        $ 4528 "Until (tool_contact_detection)"
        break
      end
      sync()
    end
    $ 4529 "Direction: Base Z+"
    global move_thread_flag_4529=0
    thread move_thread_4529():
      enter_critical
      move_thread_flag_4529 = 1
      local towardsPos=calculate_point_to_move_towards(p[0.0,0.0,0.0,0.0,0.0,0.0], [0.0,0.0,1.0], 0.08)
      movel(towardsPos, a=0.15, v=0.1)
      move_thread_flag_4529 = 2
      exit_critical
    end
    move_thread_flag_4529 = 0
    move_thread_han_4529 = run move_thread_4529()
    while (True):
      sleep(1.0E-10)
      if (move_thread_flag_4529 > 1):
        join move_thread_han_4529
        $ 4530 "Until (distance)"
        break
      end
      sync()
    end
    $ 4531 "AB"
    $ 4532 "'desbaste_inicial'"
    # 'desbaste_inicial'
    $ 4533 "bajada_broca≔p[0,0,-0.008,0,0,0]"
    global bajada_broca=p[0,0,-0.008,0,0,0]
    $ 4534 "barrenos_menos1≔2"
    global barrenos_menos1=2
    $ 4535 "barreno_actual≔0"
    global barreno_actual=0
    $ 4536 "Loop barreno_actual≤barrenos_menos1"
    while (barreno_actual <= barrenos_menos1):
      $ 4537 "Perforacion"
      $ 4538 "MoveL"
      $ 4541 "internos≔interpolate_pose(Linea25_A, Linea25_B, barreno_actual/barrenos_menos1)"
      global internos= interpolate_pose (Linea25_A_p, Linea25_B_p, barreno_actual/barrenos_menos1)
      $ 4542 "internos" "breakAfter"
      movel(internos, a=0.5, v=0.1)
      $ 4543 "'desbaste_inicial'"
      # 'desbaste_inicial'
      $ 4544 "bajada_broca≔p[0,0,-0.024,0,0,0]"
      global bajada_broca=p[0,0,-0.024,0,0,0]
      $ 4545 "bajada≔p[0,0,0.024,0,0,0]"
      global bajada=p[0,0,0.024,0,0,0]
      $ 4546 "Direction: Base Z-"
      global move_thread_flag_4546=0
      thread move_thread_4546():
        enter_critical
        move_thread_flag_4546 = 1
        local towardsPos=calculate_point_to_move_towards(p[0.0,0.0,0.0,0.0,0.0,0.0], [0.0,0.0,-1.0], 0.071)
        movel(towardsPos, a=0.15, v=0.1)
        move_thread_flag_4546 = 2
        exit_critical
      end
      move_thread_flag_4546 = 0
      move_thread_han_4546 = run move_thread_4546()
      while (True):
        sleep(1.0E-10)
        if (move_thread_flag_4546 > 1):
          join move_thread_han_4546
          $ 4547 "Until (distance)"
          break
        end
        sync()
      end
      $ 4548 "Direction: Base Z-"
      global move_thread_flag_4548=0
      thread move_thread_4548():
        enter_critical
        move_thread_flag_4548 = 1
        local towardsPos=calculate_point_to_move_towards(p[0.0,0.0,0.0,0.0,0.0,0.0], [0.0,0.0,-1.0], 1000.0)
        movel(towardsPos, a=0.007, v=0.007)
        move_thread_flag_4548 = 2
        exit_critical
      end
      move_thread_flag_4548 = 0
      move_thread_han_4548 = run move_thread_4548()
      while (True):
        local targetTcpDirection=get_target_tcp_speed()
        local stepsToRetract=tool_contact(direction=targetTcpDirection)
        if (stepsToRetract > 0):
          kill move_thread_han_4548
          stopl(0.02)
          local backTrackMovement=get_actual_joint_positions_history(stepsToRetract)
          local contactPose=get_forward_kin(backTrackMovement)
          local posDir=[targetTcpDirection[0],targetTcpDirection[1],targetTcpDirection[2]]
          local retractTo=contactPose
          if (norm(posDir) > 1e-6):
            local normalizedPosDir=normalize(posDir)
            local additionalRetraction=p[normalizedPosDir[0] * 0.0, normalizedPosDir[1] * 0.0, normalizedPosDir[2] * 0.0, 0, 0, 0]
            retractTo = pose_sub(contactPose, additionalRetraction)
          end
          movel(retractTo, a=0.02, v=0.1)
          $ 4549 "Until (tool_contact_detection)"
          break
        end
        sync()
      end
      $ 4550 "Popup: punto contacto alanzdo"
      popup("punto contacto alanzdo", "Mensaje", False, False, blocking=True)
      $ 4551 "Direction: Base Z+"
      global move_thread_flag_4551=0
      thread move_thread_4551():
        enter_critical
        move_thread_flag_4551 = 1
        local towardsPos=calculate_point_to_move_towards(p[0.0,0.0,0.0,0.0,0.0,0.0], [0.0,0.0,1.0], 0.007)
        movel(towardsPos, a=0.015, v=0.015)
        move_thread_flag_4551 = 2
        exit_critical
      end
      move_thread_flag_4551 = 0
      move_thread_han_4551 = run move_thread_4551()
      while (True):
        sleep(1.0E-10)
        if (move_thread_flag_4551 > 1):
          join move_thread_han_4551
          $ 4552 "Until (distance)"
          break
        end
        sync()
      end
      $ 4553 "Wait: 0.3"
      sleep(0.3)
      $ 4554 "Set CO[1]=Encender"
      set_configurable_digital_out(1, True)
      $ 4555 "Wait: 0.3"
      sleep(0.3)
      $ 4556 "Loop 1 times"
      Loop_135 = 0
      while (Loop_135 < 1):
        $ 4557 "bajar≔pose_add(get_actual_tcp_pose(), bajada_broca)"
        global bajar= pose_add ( get_actual_tcp_pose (), bajada_broca)
        $ 4558 "bajar" "breakAfter"
        movel(bajar, a=0.004, v=0.004)
        $ 4559 "subir≔pose_sub(get_actual_tcp_pose(), bajada_broca)"
        global subir= pose_sub ( get_actual_tcp_pose (), bajada_broca)
        $ 4560 "Direction: Base Z+"
        global move_thread_flag_4560=0
        thread move_thread_4560():
          enter_critical
          move_thread_flag_4560 = 1
          local towardsPos=calculate_point_to_move_towards(p[0.0,0.0,0.0,0.0,0.0,0.0], [0.0,0.0,1.0], 0.002)
          movel(towardsPos, a=0.015, v=0.015)
          move_thread_flag_4560 = 2
          exit_critical
        end
        move_thread_flag_4560 = 0
        move_thread_han_4560 = run move_thread_4560()
        while (True):
          sleep(1.0E-10)
          if (move_thread_flag_4560 > 1):
            join move_thread_han_4560
            $ 4561 "Until (distance)"
            break
          end
          sync()
        end
        $ 4562 "Set CO[1]=Apagar"
        set_configurable_digital_out(1, False)
        $ 4563 "subir" "breakAfter"
        movel(subir, a=0.015, v=0.015)
        $ 4564 "bajada_broca≔pose_sub(bajada_broca, bajada)"
        global bajada_broca= pose_sub (bajada_broca, bajada)
        Loop_135 = Loop_135 + 1
      end
      $ 4565 "Direction: Base Z+"
      global move_thread_flag_4565=0
      thread move_thread_4565():
        enter_critical
        move_thread_flag_4565 = 1
        local towardsPos=calculate_point_to_move_towards(p[0.0,0.0,0.0,0.0,0.0,0.0], [0.0,0.0,1.0], 0.08)
        movel(towardsPos, a=0.15, v=0.1)
        move_thread_flag_4565 = 2
        exit_critical
      end
      move_thread_flag_4565 = 0
      move_thread_han_4565 = run move_thread_4565()
      while (True):
        sleep(1.0E-10)
        if (move_thread_flag_4565 > 1):
          join move_thread_han_4565
          $ 4566 "Until (distance)"
          break
        end
        sync()
      end
      $ 4567 "Set CO[1]=Apagar"
      set_configurable_digital_out(1, False)
      $ 4568 "barreno_actual≔barreno_actual+1"
      global barreno_actual=barreno_actual+1
    end
    $ 4571 "Popup: Linea25 con chica Terminada!"
    popup("Linea25 con chica Terminada!", "Mensaje", False, False, blocking=True)
    $ 4572 "Linea26"
    $ 4573 "Marcar_puntos"
    $ 4574 "MoveL"
    $ 4575 "Linea26_A" "breakAfter"
    movel(Linea26_A_p, a=0.5, v=0.1)
    $ 4576 "bajada_comprobacion"
    $ 4577 "Direction: Base Z-"
    global move_thread_flag_4577=0
    thread move_thread_4577():
      enter_critical
      move_thread_flag_4577 = 1
      local towardsPos=calculate_point_to_move_towards(p[0.0,0.0,0.0,0.0,0.0,0.0], [0.0,0.0,-1.0], 0.071)
      movel(towardsPos, a=0.15, v=0.1)
      move_thread_flag_4577 = 2
      exit_critical
    end
    move_thread_flag_4577 = 0
    move_thread_han_4577 = run move_thread_4577()
    while (True):
      sleep(1.0E-10)
      if (move_thread_flag_4577 > 1):
        join move_thread_han_4577
        $ 4578 "Until (distance)"
        break
      end
      sync()
    end
    $ 4579 "Direction: Base Z-"
    global move_thread_flag_4579=0
    thread move_thread_4579():
      enter_critical
      move_thread_flag_4579 = 1
      local towardsPos=calculate_point_to_move_towards(p[0.0,0.0,0.0,0.0,0.0,0.0], [0.0,0.0,-1.0], 1000.0)
      movel(towardsPos, a=0.007, v=0.007)
      move_thread_flag_4579 = 2
      exit_critical
    end
    move_thread_flag_4579 = 0
    move_thread_han_4579 = run move_thread_4579()
    while (True):
      local targetTcpDirection=get_target_tcp_speed()
      local stepsToRetract=tool_contact(direction=targetTcpDirection)
      if (stepsToRetract > 0):
        kill move_thread_han_4579
        stopl(0.02)
        local backTrackMovement=get_actual_joint_positions_history(stepsToRetract)
        local contactPose=get_forward_kin(backTrackMovement)
        local posDir=[targetTcpDirection[0],targetTcpDirection[1],targetTcpDirection[2]]
        local retractTo=contactPose
        if (norm(posDir) > 1e-6):
          local normalizedPosDir=normalize(posDir)
          local additionalRetraction=p[normalizedPosDir[0] * 0.0, normalizedPosDir[1] * 0.0, normalizedPosDir[2] * 0.0, 0, 0, 0]
          retractTo = pose_sub(contactPose, additionalRetraction)
        end
        movel(retractTo, a=0.02, v=0.1)
        $ 4580 "Until (tool_contact_detection)"
        break
      end
      sync()
    end
    $ 4581 "Direction: Base Z+"
    global move_thread_flag_4581=0
    thread move_thread_4581():
      enter_critical
      move_thread_flag_4581 = 1
      local towardsPos=calculate_point_to_move_towards(p[0.0,0.0,0.0,0.0,0.0,0.0], [0.0,0.0,1.0], 0.08)
      movel(towardsPos, a=0.15, v=0.1)
      move_thread_flag_4581 = 2
      exit_critical
    end
    move_thread_flag_4581 = 0
    move_thread_han_4581 = run move_thread_4581()
    while (True):
      sleep(1.0E-10)
      if (move_thread_flag_4581 > 1):
        join move_thread_han_4581
        $ 4582 "Until (distance)"
        break
      end
      sync()
    end
    $ 4583 "Linea26_B" "breakAfter"
    movel(Linea26_B_p, a=0.5, v=0.1)
    $ 4584 "bajada_comprobacion"
    $ 4585 "Direction: Base Z-"
    global move_thread_flag_4585=0
    thread move_thread_4585():
      enter_critical
      move_thread_flag_4585 = 1
      local towardsPos=calculate_point_to_move_towards(p[0.0,0.0,0.0,0.0,0.0,0.0], [0.0,0.0,-1.0], 0.071)
      movel(towardsPos, a=0.15, v=0.1)
      move_thread_flag_4585 = 2
      exit_critical
    end
    move_thread_flag_4585 = 0
    move_thread_han_4585 = run move_thread_4585()
    while (True):
      sleep(1.0E-10)
      if (move_thread_flag_4585 > 1):
        join move_thread_han_4585
        $ 4586 "Until (distance)"
        break
      end
      sync()
    end
    $ 4587 "Direction: Base Z-"
    global move_thread_flag_4587=0
    thread move_thread_4587():
      enter_critical
      move_thread_flag_4587 = 1
      local towardsPos=calculate_point_to_move_towards(p[0.0,0.0,0.0,0.0,0.0,0.0], [0.0,0.0,-1.0], 1000.0)
      movel(towardsPos, a=0.007, v=0.007)
      move_thread_flag_4587 = 2
      exit_critical
    end
    move_thread_flag_4587 = 0
    move_thread_han_4587 = run move_thread_4587()
    while (True):
      local targetTcpDirection=get_target_tcp_speed()
      local stepsToRetract=tool_contact(direction=targetTcpDirection)
      if (stepsToRetract > 0):
        kill move_thread_han_4587
        stopl(0.02)
        local backTrackMovement=get_actual_joint_positions_history(stepsToRetract)
        local contactPose=get_forward_kin(backTrackMovement)
        local posDir=[targetTcpDirection[0],targetTcpDirection[1],targetTcpDirection[2]]
        local retractTo=contactPose
        if (norm(posDir) > 1e-6):
          local normalizedPosDir=normalize(posDir)
          local additionalRetraction=p[normalizedPosDir[0] * 0.0, normalizedPosDir[1] * 0.0, normalizedPosDir[2] * 0.0, 0, 0, 0]
          retractTo = pose_sub(contactPose, additionalRetraction)
        end
        movel(retractTo, a=0.02, v=0.1)
        $ 4588 "Until (tool_contact_detection)"
        break
      end
      sync()
    end
    $ 4589 "Direction: Base Z+"
    global move_thread_flag_4589=0
    thread move_thread_4589():
      enter_critical
      move_thread_flag_4589 = 1
      local towardsPos=calculate_point_to_move_towards(p[0.0,0.0,0.0,0.0,0.0,0.0], [0.0,0.0,1.0], 0.08)
      movel(towardsPos, a=0.15, v=0.1)
      move_thread_flag_4589 = 2
      exit_critical
    end
    move_thread_flag_4589 = 0
    move_thread_han_4589 = run move_thread_4589()
    while (True):
      sleep(1.0E-10)
      if (move_thread_flag_4589 > 1):
        join move_thread_han_4589
        $ 4590 "Until (distance)"
        break
      end
      sync()
    end
    $ 4591 "AB"
    $ 4592 "'desbaste_inicial'"
    # 'desbaste_inicial'
    $ 4593 "bajada_broca≔p[0,0,-0.008,0,0,0]"
    global bajada_broca=p[0,0,-0.008,0,0,0]
    $ 4594 "barrenos_menos1≔1"
    global barrenos_menos1=1
    $ 4595 "barreno_actual≔0"
    global barreno_actual=0
    $ 4596 "Loop barreno_actual≤barrenos_menos1"
    while (barreno_actual <= barrenos_menos1):
      $ 4597 "Perforacion"
      $ 4598 "MoveL"
      $ 4601 "internos≔interpolate_pose(Linea26_A, Linea26_B, barreno_actual/barrenos_menos1)"
      global internos= interpolate_pose (Linea26_A_p, Linea26_B_p, barreno_actual/barrenos_menos1)
      $ 4602 "internos" "breakAfter"
      movel(internos, a=0.5, v=0.1)
      $ 4603 "'desbaste_inicial'"
      # 'desbaste_inicial'
      $ 4604 "bajada_broca≔p[0,0,-0.024,0,0,0]"
      global bajada_broca=p[0,0,-0.024,0,0,0]
      $ 4605 "bajada≔p[0,0,0.024,0,0,0]"
      global bajada=p[0,0,0.024,0,0,0]
      $ 4606 "Direction: Base Z-"
      global move_thread_flag_4606=0
      thread move_thread_4606():
        enter_critical
        move_thread_flag_4606 = 1
        local towardsPos=calculate_point_to_move_towards(p[0.0,0.0,0.0,0.0,0.0,0.0], [0.0,0.0,-1.0], 0.071)
        movel(towardsPos, a=0.15, v=0.1)
        move_thread_flag_4606 = 2
        exit_critical
      end
      move_thread_flag_4606 = 0
      move_thread_han_4606 = run move_thread_4606()
      while (True):
        sleep(1.0E-10)
        if (move_thread_flag_4606 > 1):
          join move_thread_han_4606
          $ 4607 "Until (distance)"
          break
        end
        sync()
      end
      $ 4608 "Direction: Base Z-"
      global move_thread_flag_4608=0
      thread move_thread_4608():
        enter_critical
        move_thread_flag_4608 = 1
        local towardsPos=calculate_point_to_move_towards(p[0.0,0.0,0.0,0.0,0.0,0.0], [0.0,0.0,-1.0], 1000.0)
        movel(towardsPos, a=0.007, v=0.007)
        move_thread_flag_4608 = 2
        exit_critical
      end
      move_thread_flag_4608 = 0
      move_thread_han_4608 = run move_thread_4608()
      while (True):
        local targetTcpDirection=get_target_tcp_speed()
        local stepsToRetract=tool_contact(direction=targetTcpDirection)
        if (stepsToRetract > 0):
          kill move_thread_han_4608
          stopl(0.02)
          local backTrackMovement=get_actual_joint_positions_history(stepsToRetract)
          local contactPose=get_forward_kin(backTrackMovement)
          local posDir=[targetTcpDirection[0],targetTcpDirection[1],targetTcpDirection[2]]
          local retractTo=contactPose
          if (norm(posDir) > 1e-6):
            local normalizedPosDir=normalize(posDir)
            local additionalRetraction=p[normalizedPosDir[0] * 0.0, normalizedPosDir[1] * 0.0, normalizedPosDir[2] * 0.0, 0, 0, 0]
            retractTo = pose_sub(contactPose, additionalRetraction)
          end
          movel(retractTo, a=0.02, v=0.1)
          $ 4609 "Until (tool_contact_detection)"
          break
        end
        sync()
      end
      $ 4610 "Popup: punto contacto alanzdo"
      popup("punto contacto alanzdo", "Mensaje", False, False, blocking=True)
      $ 4611 "Direction: Base Z+"
      global move_thread_flag_4611=0
      thread move_thread_4611():
        enter_critical
        move_thread_flag_4611 = 1
        local towardsPos=calculate_point_to_move_towards(p[0.0,0.0,0.0,0.0,0.0,0.0], [0.0,0.0,1.0], 0.007)
        movel(towardsPos, a=0.015, v=0.015)
        move_thread_flag_4611 = 2
        exit_critical
      end
      move_thread_flag_4611 = 0
      move_thread_han_4611 = run move_thread_4611()
      while (True):
        sleep(1.0E-10)
        if (move_thread_flag_4611 > 1):
          join move_thread_han_4611
          $ 4612 "Until (distance)"
          break
        end
        sync()
      end
      $ 4613 "Wait: 0.3"
      sleep(0.3)
      $ 4614 "Set CO[1]=Encender"
      set_configurable_digital_out(1, True)
      $ 4615 "Wait: 0.3"
      sleep(0.3)
      $ 4616 "Loop 1 times"
      Loop_138 = 0
      while (Loop_138 < 1):
        $ 4617 "bajar≔pose_add(get_actual_tcp_pose(), bajada_broca)"
        global bajar= pose_add ( get_actual_tcp_pose (), bajada_broca)
        $ 4618 "bajar" "breakAfter"
        movel(bajar, a=0.004, v=0.004)
        $ 4619 "subir≔pose_sub(get_actual_tcp_pose(), bajada_broca)"
        global subir= pose_sub ( get_actual_tcp_pose (), bajada_broca)
        $ 4620 "Direction: Base Z+"
        global move_thread_flag_4620=0
        thread move_thread_4620():
          enter_critical
          move_thread_flag_4620 = 1
          local towardsPos=calculate_point_to_move_towards(p[0.0,0.0,0.0,0.0,0.0,0.0], [0.0,0.0,1.0], 0.002)
          movel(towardsPos, a=0.015, v=0.015)
          move_thread_flag_4620 = 2
          exit_critical
        end
        move_thread_flag_4620 = 0
        move_thread_han_4620 = run move_thread_4620()
        while (True):
          sleep(1.0E-10)
          if (move_thread_flag_4620 > 1):
            join move_thread_han_4620
            $ 4621 "Until (distance)"
            break
          end
          sync()
        end
        $ 4622 "Set CO[1]=Apagar"
        set_configurable_digital_out(1, False)
        $ 4623 "subir" "breakAfter"
        movel(subir, a=0.015, v=0.015)
        $ 4624 "bajada_broca≔pose_sub(bajada_broca, bajada)"
        global bajada_broca= pose_sub (bajada_broca, bajada)
        Loop_138 = Loop_138 + 1
      end
      $ 4625 "Direction: Base Z+"
      global move_thread_flag_4625=0
      thread move_thread_4625():
        enter_critical
        move_thread_flag_4625 = 1
        local towardsPos=calculate_point_to_move_towards(p[0.0,0.0,0.0,0.0,0.0,0.0], [0.0,0.0,1.0], 0.08)
        movel(towardsPos, a=0.15, v=0.1)
        move_thread_flag_4625 = 2
        exit_critical
      end
      move_thread_flag_4625 = 0
      move_thread_han_4625 = run move_thread_4625()
      while (True):
        sleep(1.0E-10)
        if (move_thread_flag_4625 > 1):
          join move_thread_han_4625
          $ 4626 "Until (distance)"
          break
        end
        sync()
      end
      $ 4627 "Set CO[1]=Apagar"
      set_configurable_digital_out(1, False)
      $ 4628 "barreno_actual≔barreno_actual+1"
      global barreno_actual=barreno_actual+1
    end
    $ 4631 "Popup: Linea26 con chica Terminada!"
    popup("Linea26 con chica Terminada!", "Mensaje", False, False, blocking=True)
    $ 4632 "Linea27"
    $ 4633 "Marcar_puntos"
    $ 4634 "MoveL"
    $ 4635 "Linea27_A" "breakAfter"
    movel(Linea27_A_p, a=0.5, v=0.1)
    $ 4636 "bajada_comprobacion"
    $ 4637 "Direction: Base Z-"
    global move_thread_flag_4637=0
    thread move_thread_4637():
      enter_critical
      move_thread_flag_4637 = 1
      local towardsPos=calculate_point_to_move_towards(p[0.0,0.0,0.0,0.0,0.0,0.0], [0.0,0.0,-1.0], 0.071)
      movel(towardsPos, a=0.15, v=0.1)
      move_thread_flag_4637 = 2
      exit_critical
    end
    move_thread_flag_4637 = 0
    move_thread_han_4637 = run move_thread_4637()
    while (True):
      sleep(1.0E-10)
      if (move_thread_flag_4637 > 1):
        join move_thread_han_4637
        $ 4638 "Until (distance)"
        break
      end
      sync()
    end
    $ 4639 "Direction: Base Z-"
    global move_thread_flag_4639=0
    thread move_thread_4639():
      enter_critical
      move_thread_flag_4639 = 1
      local towardsPos=calculate_point_to_move_towards(p[0.0,0.0,0.0,0.0,0.0,0.0], [0.0,0.0,-1.0], 1000.0)
      movel(towardsPos, a=0.007, v=0.007)
      move_thread_flag_4639 = 2
      exit_critical
    end
    move_thread_flag_4639 = 0
    move_thread_han_4639 = run move_thread_4639()
    while (True):
      local targetTcpDirection=get_target_tcp_speed()
      local stepsToRetract=tool_contact(direction=targetTcpDirection)
      if (stepsToRetract > 0):
        kill move_thread_han_4639
        stopl(0.02)
        local backTrackMovement=get_actual_joint_positions_history(stepsToRetract)
        local contactPose=get_forward_kin(backTrackMovement)
        local posDir=[targetTcpDirection[0],targetTcpDirection[1],targetTcpDirection[2]]
        local retractTo=contactPose
        if (norm(posDir) > 1e-6):
          local normalizedPosDir=normalize(posDir)
          local additionalRetraction=p[normalizedPosDir[0] * 0.0, normalizedPosDir[1] * 0.0, normalizedPosDir[2] * 0.0, 0, 0, 0]
          retractTo = pose_sub(contactPose, additionalRetraction)
        end
        movel(retractTo, a=0.02, v=0.1)
        $ 4640 "Until (tool_contact_detection)"
        break
      end
      sync()
    end
    $ 4641 "Direction: Base Z+"
    global move_thread_flag_4641=0
    thread move_thread_4641():
      enter_critical
      move_thread_flag_4641 = 1
      local towardsPos=calculate_point_to_move_towards(p[0.0,0.0,0.0,0.0,0.0,0.0], [0.0,0.0,1.0], 0.08)
      movel(towardsPos, a=0.15, v=0.1)
      move_thread_flag_4641 = 2
      exit_critical
    end
    move_thread_flag_4641 = 0
    move_thread_han_4641 = run move_thread_4641()
    while (True):
      sleep(1.0E-10)
      if (move_thread_flag_4641 > 1):
        join move_thread_han_4641
        $ 4642 "Until (distance)"
        break
      end
      sync()
    end
    $ 4643 "Linea27_B" "breakAfter"
    movel(Linea27_B_p, a=0.5, v=0.1)
    $ 4644 "bajada_comprobacion"
    $ 4645 "Direction: Base Z-"
    global move_thread_flag_4645=0
    thread move_thread_4645():
      enter_critical
      move_thread_flag_4645 = 1
      local towardsPos=calculate_point_to_move_towards(p[0.0,0.0,0.0,0.0,0.0,0.0], [0.0,0.0,-1.0], 0.071)
      movel(towardsPos, a=0.15, v=0.1)
      move_thread_flag_4645 = 2
      exit_critical
    end
    move_thread_flag_4645 = 0
    move_thread_han_4645 = run move_thread_4645()
    while (True):
      sleep(1.0E-10)
      if (move_thread_flag_4645 > 1):
        join move_thread_han_4645
        $ 4646 "Until (distance)"
        break
      end
      sync()
    end
    $ 4647 "Direction: Base Z-"
    global move_thread_flag_4647=0
    thread move_thread_4647():
      enter_critical
      move_thread_flag_4647 = 1
      local towardsPos=calculate_point_to_move_towards(p[0.0,0.0,0.0,0.0,0.0,0.0], [0.0,0.0,-1.0], 1000.0)
      movel(towardsPos, a=0.007, v=0.007)
      move_thread_flag_4647 = 2
      exit_critical
    end
    move_thread_flag_4647 = 0
    move_thread_han_4647 = run move_thread_4647()
    while (True):
      local targetTcpDirection=get_target_tcp_speed()
      local stepsToRetract=tool_contact(direction=targetTcpDirection)
      if (stepsToRetract > 0):
        kill move_thread_han_4647
        stopl(0.02)
        local backTrackMovement=get_actual_joint_positions_history(stepsToRetract)
        local contactPose=get_forward_kin(backTrackMovement)
        local posDir=[targetTcpDirection[0],targetTcpDirection[1],targetTcpDirection[2]]
        local retractTo=contactPose
        if (norm(posDir) > 1e-6):
          local normalizedPosDir=normalize(posDir)
          local additionalRetraction=p[normalizedPosDir[0] * 0.0, normalizedPosDir[1] * 0.0, normalizedPosDir[2] * 0.0, 0, 0, 0]
          retractTo = pose_sub(contactPose, additionalRetraction)
        end
        movel(retractTo, a=0.02, v=0.1)
        $ 4648 "Until (tool_contact_detection)"
        break
      end
      sync()
    end
    $ 4649 "Direction: Base Z+"
    global move_thread_flag_4649=0
    thread move_thread_4649():
      enter_critical
      move_thread_flag_4649 = 1
      local towardsPos=calculate_point_to_move_towards(p[0.0,0.0,0.0,0.0,0.0,0.0], [0.0,0.0,1.0], 0.08)
      movel(towardsPos, a=0.15, v=0.1)
      move_thread_flag_4649 = 2
      exit_critical
    end
    move_thread_flag_4649 = 0
    move_thread_han_4649 = run move_thread_4649()
    while (True):
      sleep(1.0E-10)
      if (move_thread_flag_4649 > 1):
        join move_thread_han_4649
        $ 4650 "Until (distance)"
        break
      end
      sync()
    end
    $ 4651 "AB"
    $ 4652 "'desbaste_inicial'"
    # 'desbaste_inicial'
    $ 4653 "bajada_broca≔p[0,0,-0.008,0,0,0]"
    global bajada_broca=p[0,0,-0.008,0,0,0]
    $ 4654 "barrenos_menos1≔6"
    global barrenos_menos1=6
    $ 4655 "barreno_actual≔0"
    global barreno_actual=0
    $ 4656 "Loop barreno_actual≤barrenos_menos1"
    while (barreno_actual <= barrenos_menos1):
      $ 4657 "Perforacion"
      $ 4658 "MoveL"
      $ 4659 "If barreno_actual≟3"
      if (barreno_actual == 3):
        $ 4660 "barreno_actual≔barreno_actual+1"
        global barreno_actual=barreno_actual+1
      end
      $ 4661 "internos≔interpolate_pose(Linea27_A, Linea27_B, barreno_actual/barrenos_menos1)"
      global internos= interpolate_pose (Linea27_A_p, Linea27_B_p, barreno_actual/barrenos_menos1)
      $ 4662 "internos" "breakAfter"
      movel(internos, a=0.5, v=0.1)
      $ 4663 "'desbaste_inicial'"
      # 'desbaste_inicial'
      $ 4664 "bajada_broca≔p[0,0,-0.024,0,0,0]"
      global bajada_broca=p[0,0,-0.024,0,0,0]
      $ 4665 "bajada≔p[0,0,0.024,0,0,0]"
      global bajada=p[0,0,0.024,0,0,0]
      $ 4666 "Direction: Base Z-"
      global move_thread_flag_4666=0
      thread move_thread_4666():
        enter_critical
        move_thread_flag_4666 = 1
        local towardsPos=calculate_point_to_move_towards(p[0.0,0.0,0.0,0.0,0.0,0.0], [0.0,0.0,-1.0], 0.071)
        movel(towardsPos, a=0.15, v=0.1)
        move_thread_flag_4666 = 2
        exit_critical
      end
      move_thread_flag_4666 = 0
      move_thread_han_4666 = run move_thread_4666()
      while (True):
        sleep(1.0E-10)
        if (move_thread_flag_4666 > 1):
          join move_thread_han_4666
          $ 4667 "Until (distance)"
          break
        end
        sync()
      end
      $ 4668 "Direction: Base Z-"
      global move_thread_flag_4668=0
      thread move_thread_4668():
        enter_critical
        move_thread_flag_4668 = 1
        local towardsPos=calculate_point_to_move_towards(p[0.0,0.0,0.0,0.0,0.0,0.0], [0.0,0.0,-1.0], 1000.0)
        movel(towardsPos, a=0.007, v=0.007)
        move_thread_flag_4668 = 2
        exit_critical
      end
      move_thread_flag_4668 = 0
      move_thread_han_4668 = run move_thread_4668()
      while (True):
        local targetTcpDirection=get_target_tcp_speed()
        local stepsToRetract=tool_contact(direction=targetTcpDirection)
        if (stepsToRetract > 0):
          kill move_thread_han_4668
          stopl(0.02)
          local backTrackMovement=get_actual_joint_positions_history(stepsToRetract)
          local contactPose=get_forward_kin(backTrackMovement)
          local posDir=[targetTcpDirection[0],targetTcpDirection[1],targetTcpDirection[2]]
          local retractTo=contactPose
          if (norm(posDir) > 1e-6):
            local normalizedPosDir=normalize(posDir)
            local additionalRetraction=p[normalizedPosDir[0] * 0.0, normalizedPosDir[1] * 0.0, normalizedPosDir[2] * 0.0, 0, 0, 0]
            retractTo = pose_sub(contactPose, additionalRetraction)
          end
          movel(retractTo, a=0.02, v=0.1)
          $ 4669 "Until (tool_contact_detection)"
          break
        end
        sync()
      end
      $ 4670 "Popup: punto contacto alanzdo"
      popup("punto contacto alanzdo", "Mensaje", False, False, blocking=True)
      $ 4671 "Direction: Base Z+"
      global move_thread_flag_4671=0
      thread move_thread_4671():
        enter_critical
        move_thread_flag_4671 = 1
        local towardsPos=calculate_point_to_move_towards(p[0.0,0.0,0.0,0.0,0.0,0.0], [0.0,0.0,1.0], 0.007)
        movel(towardsPos, a=0.015, v=0.015)
        move_thread_flag_4671 = 2
        exit_critical
      end
      move_thread_flag_4671 = 0
      move_thread_han_4671 = run move_thread_4671()
      while (True):
        sleep(1.0E-10)
        if (move_thread_flag_4671 > 1):
          join move_thread_han_4671
          $ 4672 "Until (distance)"
          break
        end
        sync()
      end
      $ 4673 "Wait: 0.3"
      sleep(0.3)
      $ 4674 "Set CO[1]=Encender"
      set_configurable_digital_out(1, True)
      $ 4675 "Wait: 0.3"
      sleep(0.3)
      $ 4676 "Loop 1 times"
      Loop_142 = 0
      while (Loop_142 < 1):
        $ 4677 "bajar≔pose_add(get_actual_tcp_pose(), bajada_broca)"
        global bajar= pose_add ( get_actual_tcp_pose (), bajada_broca)
        $ 4678 "bajar" "breakAfter"
        movel(bajar, a=0.004, v=0.004)
        $ 4679 "subir≔pose_sub(get_actual_tcp_pose(), bajada_broca)"
        global subir= pose_sub ( get_actual_tcp_pose (), bajada_broca)
        $ 4680 "Direction: Base Z+"
        global move_thread_flag_4680=0
        thread move_thread_4680():
          enter_critical
          move_thread_flag_4680 = 1
          local towardsPos=calculate_point_to_move_towards(p[0.0,0.0,0.0,0.0,0.0,0.0], [0.0,0.0,1.0], 0.002)
          movel(towardsPos, a=0.015, v=0.015)
          move_thread_flag_4680 = 2
          exit_critical
        end
        move_thread_flag_4680 = 0
        move_thread_han_4680 = run move_thread_4680()
        while (True):
          sleep(1.0E-10)
          if (move_thread_flag_4680 > 1):
            join move_thread_han_4680
            $ 4681 "Until (distance)"
            break
          end
          sync()
        end
        $ 4682 "Set CO[1]=Apagar"
        set_configurable_digital_out(1, False)
        $ 4683 "subir" "breakAfter"
        movel(subir, a=0.015, v=0.015)
        $ 4684 "bajada_broca≔pose_sub(bajada_broca, bajada)"
        global bajada_broca= pose_sub (bajada_broca, bajada)
        Loop_142 = Loop_142 + 1
      end
      $ 4685 "Direction: Base Z+"
      global move_thread_flag_4685=0
      thread move_thread_4685():
        enter_critical
        move_thread_flag_4685 = 1
        local towardsPos=calculate_point_to_move_towards(p[0.0,0.0,0.0,0.0,0.0,0.0], [0.0,0.0,1.0], 0.08)
        movel(towardsPos, a=0.15, v=0.1)
        move_thread_flag_4685 = 2
        exit_critical
      end
      move_thread_flag_4685 = 0
      move_thread_han_4685 = run move_thread_4685()
      while (True):
        sleep(1.0E-10)
        if (move_thread_flag_4685 > 1):
          join move_thread_han_4685
          $ 4686 "Until (distance)"
          break
        end
        sync()
      end
      $ 4687 "Set CO[1]=Apagar"
      set_configurable_digital_out(1, False)
      $ 4688 "barreno_actual≔barreno_actual+1"
      global barreno_actual=barreno_actual+1
    end
    $ 4691 "Popup: Linea27 con chica Terminada!"
    popup("Linea27 con chica Terminada!", "Mensaje", False, False, blocking=True)
    $ 4692 "Linea28"
    $ 4693 "Marcar_puntos"
    $ 4694 "MoveL"
    $ 4695 "Linea28_B" "breakAfter"
    movel(Linea28_B_p, a=0.5, v=0.1)
    $ 4696 "bajada_comprobacion"
    $ 4697 "Direction: Base Z-"
    global move_thread_flag_4697=0
    thread move_thread_4697():
      enter_critical
      move_thread_flag_4697 = 1
      local towardsPos=calculate_point_to_move_towards(p[0.0,0.0,0.0,0.0,0.0,0.0], [0.0,0.0,-1.0], 0.071)
      movel(towardsPos, a=0.15, v=0.1)
      move_thread_flag_4697 = 2
      exit_critical
    end
    move_thread_flag_4697 = 0
    move_thread_han_4697 = run move_thread_4697()
    while (True):
      sleep(1.0E-10)
      if (move_thread_flag_4697 > 1):
        join move_thread_han_4697
        $ 4698 "Until (distance)"
        break
      end
      sync()
    end
    $ 4699 "Direction: Base Z-"
    global move_thread_flag_4699=0
    thread move_thread_4699():
      enter_critical
      move_thread_flag_4699 = 1
      local towardsPos=calculate_point_to_move_towards(p[0.0,0.0,0.0,0.0,0.0,0.0], [0.0,0.0,-1.0], 1000.0)
      movel(towardsPos, a=0.007, v=0.007)
      move_thread_flag_4699 = 2
      exit_critical
    end
    move_thread_flag_4699 = 0
    move_thread_han_4699 = run move_thread_4699()
    while (True):
      local targetTcpDirection=get_target_tcp_speed()
      local stepsToRetract=tool_contact(direction=targetTcpDirection)
      if (stepsToRetract > 0):
        kill move_thread_han_4699
        stopl(0.02)
        local backTrackMovement=get_actual_joint_positions_history(stepsToRetract)
        local contactPose=get_forward_kin(backTrackMovement)
        local posDir=[targetTcpDirection[0],targetTcpDirection[1],targetTcpDirection[2]]
        local retractTo=contactPose
        if (norm(posDir) > 1e-6):
          local normalizedPosDir=normalize(posDir)
          local additionalRetraction=p[normalizedPosDir[0] * 0.0, normalizedPosDir[1] * 0.0, normalizedPosDir[2] * 0.0, 0, 0, 0]
          retractTo = pose_sub(contactPose, additionalRetraction)
        end
        movel(retractTo, a=0.02, v=0.1)
        $ 4700 "Until (tool_contact_detection)"
        break
      end
      sync()
    end
    $ 4701 "Direction: Base Z+"
    global move_thread_flag_4701=0
    thread move_thread_4701():
      enter_critical
      move_thread_flag_4701 = 1
      local towardsPos=calculate_point_to_move_towards(p[0.0,0.0,0.0,0.0,0.0,0.0], [0.0,0.0,1.0], 0.08)
      movel(towardsPos, a=0.15, v=0.1)
      move_thread_flag_4701 = 2
      exit_critical
    end
    move_thread_flag_4701 = 0
    move_thread_han_4701 = run move_thread_4701()
    while (True):
      sleep(1.0E-10)
      if (move_thread_flag_4701 > 1):
        join move_thread_han_4701
        $ 4702 "Until (distance)"
        break
      end
      sync()
    end
    $ 4703 "AB"
    $ 4704 "'desbaste_inicial'"
    # 'desbaste_inicial'
    $ 4705 "bajada_broca≔p[0,0,-0.008,0,0,0]"
    global bajada_broca=p[0,0,-0.008,0,0,0]
    $ 4706 "barrenos_menos1≔0"
    global barrenos_menos1=0
    $ 4707 "barreno_actual≔0"
    global barreno_actual=0
    $ 4708 "Loop barreno_actual≤barrenos_menos1"
    while (barreno_actual <= barrenos_menos1):
      $ 4709 "Perforacion"
      $ 4710 "MoveL"
      $ 4715 "Linea28_B" "breakAfter"
      movel(Linea28_B_p, a=0.5, v=0.1)
      $ 4716 "'desbaste_inicial'"
      # 'desbaste_inicial'
      $ 4717 "bajada_broca≔p[0,0,-0.024,0,0,0]"
      global bajada_broca=p[0,0,-0.024,0,0,0]
      $ 4718 "bajada≔p[0,0,0.024,0,0,0]"
      global bajada=p[0,0,0.024,0,0,0]
      $ 4719 "Direction: Base Z-"
      global move_thread_flag_4719=0
      thread move_thread_4719():
        enter_critical
        move_thread_flag_4719 = 1
        local towardsPos=calculate_point_to_move_towards(p[0.0,0.0,0.0,0.0,0.0,0.0], [0.0,0.0,-1.0], 0.071)
        movel(towardsPos, a=0.15, v=0.1)
        move_thread_flag_4719 = 2
        exit_critical
      end
      move_thread_flag_4719 = 0
      move_thread_han_4719 = run move_thread_4719()
      while (True):
        sleep(1.0E-10)
        if (move_thread_flag_4719 > 1):
          join move_thread_han_4719
          $ 4720 "Until (distance)"
          break
        end
        sync()
      end
      $ 4721 "Direction: Base Z-"
      global move_thread_flag_4721=0
      thread move_thread_4721():
        enter_critical
        move_thread_flag_4721 = 1
        local towardsPos=calculate_point_to_move_towards(p[0.0,0.0,0.0,0.0,0.0,0.0], [0.0,0.0,-1.0], 1000.0)
        movel(towardsPos, a=0.007, v=0.007)
        move_thread_flag_4721 = 2
        exit_critical
      end
      move_thread_flag_4721 = 0
      move_thread_han_4721 = run move_thread_4721()
      while (True):
        local targetTcpDirection=get_target_tcp_speed()
        local stepsToRetract=tool_contact(direction=targetTcpDirection)
        if (stepsToRetract > 0):
          kill move_thread_han_4721
          stopl(0.02)
          local backTrackMovement=get_actual_joint_positions_history(stepsToRetract)
          local contactPose=get_forward_kin(backTrackMovement)
          local posDir=[targetTcpDirection[0],targetTcpDirection[1],targetTcpDirection[2]]
          local retractTo=contactPose
          if (norm(posDir) > 1e-6):
            local normalizedPosDir=normalize(posDir)
            local additionalRetraction=p[normalizedPosDir[0] * 0.0, normalizedPosDir[1] * 0.0, normalizedPosDir[2] * 0.0, 0, 0, 0]
            retractTo = pose_sub(contactPose, additionalRetraction)
          end
          movel(retractTo, a=0.02, v=0.1)
          $ 4722 "Until (tool_contact_detection)"
          break
        end
        sync()
      end
      $ 4723 "Popup: punto contacto alanzdo"
      popup("punto contacto alanzdo", "Mensaje", False, False, blocking=True)
      $ 4724 "Direction: Base Z+"
      global move_thread_flag_4724=0
      thread move_thread_4724():
        enter_critical
        move_thread_flag_4724 = 1
        local towardsPos=calculate_point_to_move_towards(p[0.0,0.0,0.0,0.0,0.0,0.0], [0.0,0.0,1.0], 0.01)
        movel(towardsPos, a=0.015, v=0.015)
        move_thread_flag_4724 = 2
        exit_critical
      end
      move_thread_flag_4724 = 0
      move_thread_han_4724 = run move_thread_4724()
      while (True):
        sleep(1.0E-10)
        if (move_thread_flag_4724 > 1):
          join move_thread_han_4724
          $ 4725 "Until (distance)"
          break
        end
        sync()
      end
      $ 4726 "Wait: 0.3"
      sleep(0.3)
      $ 4727 "Set CO[1]=Encender"
      set_configurable_digital_out(1, True)
      $ 4728 "Wait: 0.3"
      sleep(0.3)
      $ 4729 "Loop 1 times"
      Loop_146 = 0
      while (Loop_146 < 1):
        $ 4730 "bajar≔pose_add(get_actual_tcp_pose(), bajada_broca)"
        global bajar= pose_add ( get_actual_tcp_pose (), bajada_broca)
        $ 4731 "bajar" "breakAfter"
        movel(bajar, a=0.004, v=0.004)
        $ 4732 "subir≔pose_sub(get_actual_tcp_pose(), bajada_broca)"
        global subir= pose_sub ( get_actual_tcp_pose (), bajada_broca)
        $ 4733 "Direction: Base Z+"
        global move_thread_flag_4733=0
        thread move_thread_4733():
          enter_critical
          move_thread_flag_4733 = 1
          local towardsPos=calculate_point_to_move_towards(p[0.0,0.0,0.0,0.0,0.0,0.0], [0.0,0.0,1.0], 0.002)
          movel(towardsPos, a=0.015, v=0.015)
          move_thread_flag_4733 = 2
          exit_critical
        end
        move_thread_flag_4733 = 0
        move_thread_han_4733 = run move_thread_4733()
        while (True):
          sleep(1.0E-10)
          if (move_thread_flag_4733 > 1):
            join move_thread_han_4733
            $ 4734 "Until (distance)"
            break
          end
          sync()
        end
        $ 4735 "Set CO[1]=Apagar"
        set_configurable_digital_out(1, False)
        $ 4736 "subir" "breakAfter"
        movel(subir, a=0.015, v=0.015)
        $ 4737 "bajada_broca≔pose_sub(bajada_broca, bajada)"
        global bajada_broca= pose_sub (bajada_broca, bajada)
        Loop_146 = Loop_146 + 1
      end
      $ 4738 "Direction: Base Z+"
      global move_thread_flag_4738=0
      thread move_thread_4738():
        enter_critical
        move_thread_flag_4738 = 1
        local towardsPos=calculate_point_to_move_towards(p[0.0,0.0,0.0,0.0,0.0,0.0], [0.0,0.0,1.0], 0.08)
        movel(towardsPos, a=0.15, v=0.1)
        move_thread_flag_4738 = 2
        exit_critical
      end
      move_thread_flag_4738 = 0
      move_thread_han_4738 = run move_thread_4738()
      while (True):
        sleep(1.0E-10)
        if (move_thread_flag_4738 > 1):
          join move_thread_han_4738
          $ 4739 "Until (distance)"
          break
        end
        sync()
      end
      $ 4740 "Set CO[1]=Apagar"
      set_configurable_digital_out(1, False)
      $ 4741 "barreno_actual≔barreno_actual+1"
      global barreno_actual=barreno_actual+1
    end
    $ 4744 "Popup: Linea28 con chica Terminada!"
    popup("Linea28 con chica Terminada!", "Mensaje", False, False, blocking=True)
    $ 4745 "Linea29"
    $ 4746 "Marcar_puntos"
    $ 4747 "MoveL"
    $ 4748 "Linea29_A" "breakAfter"
    movel(Linea29_A_p, a=0.5, v=0.1)
    $ 4750 "bajada_comprobacion"
    $ 4751 "Direction: Base Z-"
    global move_thread_flag_4751=0
    thread move_thread_4751():
      enter_critical
      move_thread_flag_4751 = 1
      local towardsPos=calculate_point_to_move_towards(p[0.0,0.0,0.0,0.0,0.0,0.0], [0.0,0.0,-1.0], 0.071)
      movel(towardsPos, a=0.15, v=0.1)
      move_thread_flag_4751 = 2
      exit_critical
    end
    move_thread_flag_4751 = 0
    move_thread_han_4751 = run move_thread_4751()
    while (True):
      sleep(1.0E-10)
      if (move_thread_flag_4751 > 1):
        join move_thread_han_4751
        $ 4752 "Until (distance)"
        break
      end
      sync()
    end
    $ 4753 "Direction: Base Z-"
    global move_thread_flag_4753=0
    thread move_thread_4753():
      enter_critical
      move_thread_flag_4753 = 1
      local towardsPos=calculate_point_to_move_towards(p[0.0,0.0,0.0,0.0,0.0,0.0], [0.0,0.0,-1.0], 1000.0)
      movel(towardsPos, a=0.007, v=0.007)
      move_thread_flag_4753 = 2
      exit_critical
    end
    move_thread_flag_4753 = 0
    move_thread_han_4753 = run move_thread_4753()
    while (True):
      local targetTcpDirection=get_target_tcp_speed()
      local stepsToRetract=tool_contact(direction=targetTcpDirection)
      if (stepsToRetract > 0):
        kill move_thread_han_4753
        stopl(0.02)
        local backTrackMovement=get_actual_joint_positions_history(stepsToRetract)
        local contactPose=get_forward_kin(backTrackMovement)
        local posDir=[targetTcpDirection[0],targetTcpDirection[1],targetTcpDirection[2]]
        local retractTo=contactPose
        if (norm(posDir) > 1e-6):
          local normalizedPosDir=normalize(posDir)
          local additionalRetraction=p[normalizedPosDir[0] * 0.0, normalizedPosDir[1] * 0.0, normalizedPosDir[2] * 0.0, 0, 0, 0]
          retractTo = pose_sub(contactPose, additionalRetraction)
        end
        movel(retractTo, a=0.02, v=0.1)
        $ 4754 "Until (tool_contact_detection)"
        break
      end
      sync()
    end
    $ 4755 "Direction: Base Z+"
    global move_thread_flag_4755=0
    thread move_thread_4755():
      enter_critical
      move_thread_flag_4755 = 1
      local towardsPos=calculate_point_to_move_towards(p[0.0,0.0,0.0,0.0,0.0,0.0], [0.0,0.0,1.0], 0.08)
      movel(towardsPos, a=0.15, v=0.1)
      move_thread_flag_4755 = 2
      exit_critical
    end
    move_thread_flag_4755 = 0
    move_thread_han_4755 = run move_thread_4755()
    while (True):
      sleep(1.0E-10)
      if (move_thread_flag_4755 > 1):
        join move_thread_han_4755
        $ 4756 "Until (distance)"
        break
      end
      sync()
    end
    $ 4758 "Linea29_AB" "breakAfter"
    movel(Linea29_AB_p, a=0.5, v=0.1)
    $ 4759 "bajada_comprobacion"
    $ 4760 "Direction: Base Z-"
    global move_thread_flag_4760=0
    thread move_thread_4760():
      enter_critical
      move_thread_flag_4760 = 1
      local towardsPos=calculate_point_to_move_towards(p[0.0,0.0,0.0,0.0,0.0,0.0], [0.0,0.0,-1.0], 0.071)
      movel(towardsPos, a=0.15, v=0.1)
      move_thread_flag_4760 = 2
      exit_critical
    end
    move_thread_flag_4760 = 0
    move_thread_han_4760 = run move_thread_4760()
    while (True):
      sleep(1.0E-10)
      if (move_thread_flag_4760 > 1):
        join move_thread_han_4760
        $ 4761 "Until (distance)"
        break
      end
      sync()
    end
    $ 4762 "Direction: Base Z-"
    global move_thread_flag_4762=0
    thread move_thread_4762():
      enter_critical
      move_thread_flag_4762 = 1
      local towardsPos=calculate_point_to_move_towards(p[0.0,0.0,0.0,0.0,0.0,0.0], [0.0,0.0,-1.0], 1000.0)
      movel(towardsPos, a=0.007, v=0.007)
      move_thread_flag_4762 = 2
      exit_critical
    end
    move_thread_flag_4762 = 0
    move_thread_han_4762 = run move_thread_4762()
    while (True):
      local targetTcpDirection=get_target_tcp_speed()
      local stepsToRetract=tool_contact(direction=targetTcpDirection)
      if (stepsToRetract > 0):
        kill move_thread_han_4762
        stopl(0.02)
        local backTrackMovement=get_actual_joint_positions_history(stepsToRetract)
        local contactPose=get_forward_kin(backTrackMovement)
        local posDir=[targetTcpDirection[0],targetTcpDirection[1],targetTcpDirection[2]]
        local retractTo=contactPose
        if (norm(posDir) > 1e-6):
          local normalizedPosDir=normalize(posDir)
          local additionalRetraction=p[normalizedPosDir[0] * 0.0, normalizedPosDir[1] * 0.0, normalizedPosDir[2] * 0.0, 0, 0, 0]
          retractTo = pose_sub(contactPose, additionalRetraction)
        end
        movel(retractTo, a=0.02, v=0.1)
        $ 4763 "Until (tool_contact_detection)"
        break
      end
      sync()
    end
    $ 4764 "Direction: Base Z+"
    global move_thread_flag_4764=0
    thread move_thread_4764():
      enter_critical
      move_thread_flag_4764 = 1
      local towardsPos=calculate_point_to_move_towards(p[0.0,0.0,0.0,0.0,0.0,0.0], [0.0,0.0,1.0], 0.08)
      movel(towardsPos, a=0.15, v=0.1)
      move_thread_flag_4764 = 2
      exit_critical
    end
    move_thread_flag_4764 = 0
    move_thread_han_4764 = run move_thread_4764()
    while (True):
      sleep(1.0E-10)
      if (move_thread_flag_4764 > 1):
        join move_thread_han_4764
        $ 4765 "Until (distance)"
        break
      end
      sync()
    end
    $ 4766 "AB"
    $ 4767 "'desbaste_inicial'"
    # 'desbaste_inicial'
    $ 4768 "bajada_broca≔p[0,0,-0.008,0,0,0]"
    global bajada_broca=p[0,0,-0.008,0,0,0]
    $ 4769 "barrenos_menos1≔9"
    global barrenos_menos1=9
    $ 4770 "barreno_actual≔0"
    global barreno_actual=0
    $ 4771 "Loop barreno_actual≤barrenos_menos1"
    while (barreno_actual <= barrenos_menos1):
      $ 4772 "Perforacion"
      $ 4773 "MoveL"
      $ 4774 "If barreno_actual≟7"
      if (barreno_actual == 7):
        $ 4775 "barreno_actual≔barreno_actual+1"
        global barreno_actual=barreno_actual+1
      end
      $ 4776 "internos≔interpolate_pose(Linea29_A, Linea29_AB, barreno_actual/barrenos_menos1)"
      global internos= interpolate_pose (Linea29_A_p, Linea29_AB_p, barreno_actual/barrenos_menos1)
      $ 4780 "internos" "breakAfter"
      movel(internos, a=0.5, v=0.1)
      $ 4781 "'desbaste_inicial'"
      # 'desbaste_inicial'
      $ 4782 "bajada_broca≔p[0,0,-0.024,0,0,0]"
      global bajada_broca=p[0,0,-0.024,0,0,0]
      $ 4783 "bajada≔p[0,0,0.024,0,0,0]"
      global bajada=p[0,0,0.024,0,0,0]
      $ 4784 "Direction: Base Z-"
      global move_thread_flag_4784=0
      thread move_thread_4784():
        enter_critical
        move_thread_flag_4784 = 1
        local towardsPos=calculate_point_to_move_towards(p[0.0,0.0,0.0,0.0,0.0,0.0], [0.0,0.0,-1.0], 0.071)
        movel(towardsPos, a=0.15, v=0.1)
        move_thread_flag_4784 = 2
        exit_critical
      end
      move_thread_flag_4784 = 0
      move_thread_han_4784 = run move_thread_4784()
      while (True):
        sleep(1.0E-10)
        if (move_thread_flag_4784 > 1):
          join move_thread_han_4784
          $ 4785 "Until (distance)"
          break
        end
        sync()
      end
      $ 4786 "Direction: Base Z-"
      global move_thread_flag_4786=0
      thread move_thread_4786():
        enter_critical
        move_thread_flag_4786 = 1
        local towardsPos=calculate_point_to_move_towards(p[0.0,0.0,0.0,0.0,0.0,0.0], [0.0,0.0,-1.0], 1000.0)
        movel(towardsPos, a=0.007, v=0.007)
        move_thread_flag_4786 = 2
        exit_critical
      end
      move_thread_flag_4786 = 0
      move_thread_han_4786 = run move_thread_4786()
      while (True):
        local targetTcpDirection=get_target_tcp_speed()
        local stepsToRetract=tool_contact(direction=targetTcpDirection)
        if (stepsToRetract > 0):
          kill move_thread_han_4786
          stopl(0.02)
          local backTrackMovement=get_actual_joint_positions_history(stepsToRetract)
          local contactPose=get_forward_kin(backTrackMovement)
          local posDir=[targetTcpDirection[0],targetTcpDirection[1],targetTcpDirection[2]]
          local retractTo=contactPose
          if (norm(posDir) > 1e-6):
            local normalizedPosDir=normalize(posDir)
            local additionalRetraction=p[normalizedPosDir[0] * 0.0, normalizedPosDir[1] * 0.0, normalizedPosDir[2] * 0.0, 0, 0, 0]
            retractTo = pose_sub(contactPose, additionalRetraction)
          end
          movel(retractTo, a=0.02, v=0.1)
          $ 4787 "Until (tool_contact_detection)"
          break
        end
        sync()
      end
      $ 4788 "Popup: punto contacto alanzdo"
      popup("punto contacto alanzdo", "Mensaje", False, False, blocking=True)
      $ 4789 "Direction: Base Z+"
      global move_thread_flag_4789=0
      thread move_thread_4789():
        enter_critical
        move_thread_flag_4789 = 1
        local towardsPos=calculate_point_to_move_towards(p[0.0,0.0,0.0,0.0,0.0,0.0], [0.0,0.0,1.0], 0.007)
        movel(towardsPos, a=0.015, v=0.015)
        move_thread_flag_4789 = 2
        exit_critical
      end
      move_thread_flag_4789 = 0
      move_thread_han_4789 = run move_thread_4789()
      while (True):
        sleep(1.0E-10)
        if (move_thread_flag_4789 > 1):
          join move_thread_han_4789
          $ 4790 "Until (distance)"
          break
        end
        sync()
      end
      $ 4791 "Wait: 0.3"
      sleep(0.3)
      $ 4792 "Set CO[1]=Encender"
      set_configurable_digital_out(1, True)
      $ 4793 "Wait: 0.3"
      sleep(0.3)
      $ 4794 "Loop 1 times"
      Loop_150 = 0
      while (Loop_150 < 1):
        $ 4795 "bajar≔pose_add(get_actual_tcp_pose(), bajada_broca)"
        global bajar= pose_add ( get_actual_tcp_pose (), bajada_broca)
        $ 4796 "bajar" "breakAfter"
        movel(bajar, a=0.004, v=0.004)
        $ 4797 "subir≔pose_sub(get_actual_tcp_pose(), bajada_broca)"
        global subir= pose_sub ( get_actual_tcp_pose (), bajada_broca)
        $ 4798 "Direction: Base Z+"
        global move_thread_flag_4798=0
        thread move_thread_4798():
          enter_critical
          move_thread_flag_4798 = 1
          local towardsPos=calculate_point_to_move_towards(p[0.0,0.0,0.0,0.0,0.0,0.0], [0.0,0.0,1.0], 0.002)
          movel(towardsPos, a=0.015, v=0.015)
          move_thread_flag_4798 = 2
          exit_critical
        end
        move_thread_flag_4798 = 0
        move_thread_han_4798 = run move_thread_4798()
        while (True):
          sleep(1.0E-10)
          if (move_thread_flag_4798 > 1):
            join move_thread_han_4798
            $ 4799 "Until (distance)"
            break
          end
          sync()
        end
        $ 4800 "Set CO[1]=Apagar"
        set_configurable_digital_out(1, False)
        $ 4801 "subir" "breakAfter"
        movel(subir, a=0.015, v=0.015)
        $ 4802 "bajada_broca≔pose_sub(bajada_broca, bajada)"
        global bajada_broca= pose_sub (bajada_broca, bajada)
        Loop_150 = Loop_150 + 1
      end
      $ 4803 "Direction: Base Z+"
      global move_thread_flag_4803=0
      thread move_thread_4803():
        enter_critical
        move_thread_flag_4803 = 1
        local towardsPos=calculate_point_to_move_towards(p[0.0,0.0,0.0,0.0,0.0,0.0], [0.0,0.0,1.0], 0.04)
        movel(towardsPos, a=0.15, v=0.1)
        move_thread_flag_4803 = 2
        exit_critical
      end
      move_thread_flag_4803 = 0
      move_thread_han_4803 = run move_thread_4803()
      while (True):
        sleep(1.0E-10)
        if (move_thread_flag_4803 > 1):
          join move_thread_han_4803
          $ 4804 "Until (distance)"
          break
        end
        sync()
      end
      $ 4805 "Set CO[1]=Apagar"
      set_configurable_digital_out(1, False)
      $ 4806 "barreno_actual≔barreno_actual+1"
      global barreno_actual=barreno_actual+1
    end
    $ 4809 "Linea29B"
    $ 4810 "Marcar_puntos"
    $ 4811 "MoveL"
    $ 4813 "Linea29_BA" "breakAfter"
    movel(Linea29_BA_p, a=0.5, v=0.1)
    $ 4814 "bajada_comprobacion"
    $ 4815 "Direction: Base Z-"
    global move_thread_flag_4815=0
    thread move_thread_4815():
      enter_critical
      move_thread_flag_4815 = 1
      local towardsPos=calculate_point_to_move_towards(p[0.0,0.0,0.0,0.0,0.0,0.0], [0.0,0.0,-1.0], 0.071)
      movel(towardsPos, a=0.15, v=0.1)
      move_thread_flag_4815 = 2
      exit_critical
    end
    move_thread_flag_4815 = 0
    move_thread_han_4815 = run move_thread_4815()
    while (True):
      sleep(1.0E-10)
      if (move_thread_flag_4815 > 1):
        join move_thread_han_4815
        $ 4816 "Until (distance)"
        break
      end
      sync()
    end
    $ 4817 "Direction: Base Z-"
    global move_thread_flag_4817=0
    thread move_thread_4817():
      enter_critical
      move_thread_flag_4817 = 1
      local towardsPos=calculate_point_to_move_towards(p[0.0,0.0,0.0,0.0,0.0,0.0], [0.0,0.0,-1.0], 1000.0)
      movel(towardsPos, a=0.007, v=0.007)
      move_thread_flag_4817 = 2
      exit_critical
    end
    move_thread_flag_4817 = 0
    move_thread_han_4817 = run move_thread_4817()
    while (True):
      local targetTcpDirection=get_target_tcp_speed()
      local stepsToRetract=tool_contact(direction=targetTcpDirection)
      if (stepsToRetract > 0):
        kill move_thread_han_4817
        stopl(0.02)
        local backTrackMovement=get_actual_joint_positions_history(stepsToRetract)
        local contactPose=get_forward_kin(backTrackMovement)
        local posDir=[targetTcpDirection[0],targetTcpDirection[1],targetTcpDirection[2]]
        local retractTo=contactPose
        if (norm(posDir) > 1e-6):
          local normalizedPosDir=normalize(posDir)
          local additionalRetraction=p[normalizedPosDir[0] * 0.0, normalizedPosDir[1] * 0.0, normalizedPosDir[2] * 0.0, 0, 0, 0]
          retractTo = pose_sub(contactPose, additionalRetraction)
        end
        movel(retractTo, a=0.02, v=0.1)
